   PRODUCT_TYPE[5].Motion.Gluing_Nozzle_Y.Position[20].Vel := 0;
   PRODUCT_TYPE[6].Motion.Gluing_Nozzle_Y.Position[20].Pos := 0.0;
   PRODUCT_TYPE[6].Motion.Gluing_Nozzle_Y.Position[20].Vel := 0;
   PRODUCT_TYPE[7].Motion.Gluing_Nozzle_Y.Position[20].Pos := 0.0;
   PRODUCT_TYPE[7].Motion.Gluing_Nozzle_Y.Position[20].Vel := 0;
   PRODUCT_TYPE[8].Motion.Gluing_Nozzle_Y.Position[20].Pos := 0.0;
   PRODUCT_TYPE[8].Motion.Gluing_Nozzle_Y.Position[20].Vel := 0;
   PRODUCT_TYPE[9].Motion.Gluing_Nozzle_Y.Position[20].Pos := 0.0;
   PRODUCT_TYPE[9].Motion.Gluing_Nozzle_Y.Position[20].Vel := 0;
   PRODUCT_TYPE[10].Motion.Gluing_Nozzle_Y.Position[20].Pos := 0.0;
   PRODUCT_TYPE[10].Motion.Gluing_Nozzle_Y.Position[20].Vel := 0;
   PRODUCT_TYPE[1].Motion.Ring_Turntable_Axis_1.Position[1].Pos := 3419;
   PRODUCT_TYPE[1].Motion.Ring_Turntable_Axis_1.Position[1].Vel := 10000;
   PRODUCT_TYPE[2].Motion.Ring_Turntable_Axis_1.Position[1].Pos := 3419;
   PRODUCT_TYPE[2].Motion.Ring_Turntable_Axis_1.Position[1].Vel := 10000;
   PRODUCT_TYPE[3].Motion.Ring_Turntable_Axis_1.Position[1].Pos := 3419;
   PRODUCT_TYPE[3].Motion.Ring_Turntable_Axis_1.Position[1].Vel := 10000;
   PRODUCT_TYPE[4].Motion.Ring_Turntable_Axis_1.Position[1].Pos := 3419;
   PRODUCT_TYPE[4].Motion.Ring_Turntable_Axis_1.Position[1].Vel := 10000;
   PRODUCT_TYPE[5].Motion.Ring_Turntable_Axis_1.Position[1].Pos := 3419;
   PRODUCT_TYPE[5].Motion.Ring_Turntable_Axis_1.Position[1].Vel := 10000;
   PRODUCT_TYPE[6].Motion.Ring_Turntable_Axis_1.Position[1].Pos := 3419;
   PRODUCT_TYPE[6].Motion.Ring_Turntable_Axis_1.Position[1].Vel := 10000;
   PRODUCT_TYPE[7].Motion.Ring_Turntable_Axis_1.Position[1].Pos := 3419;
   PRODUCT_TYPE[7].Motion.Ring_Turntable_Axis_1.Position[1].Vel := 10000;
   PRODUCT_TYPE[8].Motion.Ring_Turntable_Axis_1.Position[1].Pos := 3419;
   PRODUCT_TYPE[8].Motion.Ring_Turntable_Axis_1.Position[1].Vel := 10000;
   PRODUCT_TYPE[9].Motion.Ring_Turntable_Axis_1.Position[1].Pos := 3419;
   PRODUCT_TYPE[9].Motion.Ring_Turntable_Axis_1.Position[1].Vel := 10000;
   PRODUCT_TYPE[10].Motion.Ring_Turntable_Axis_1.Position[1].Pos := 3419;
   PRODUCT_TYPE[10].Motion.Ring_Turntable_Axis_1.Position[1].Vel := 10000;
   PRODUCT_TYPE[1].Motion.Ring_Turntable_Axis_1.Position[2].Pos := 48386;
   PRODUCT_TYPE[1].Motion.Ring_Turntable_Axis_1.Position[2].Vel := 10000;
   PRODUCT_TYPE[2].Motion.Ring_Turntable_Axis_1.Position[2].Pos := 48386;
   PRODUCT_TYPE[2].Motion.Ring_Turntable_Axis_1.Position[2].Vel := 10000;
   PRODUCT_TYPE[3].Motion.Ring_Turntable_Axis_1.Position[2].Pos := 48386;
   PRODUCT_TYPE[3].Motion.Ring_Turntable_Axis_1.Position[2].Vel := 10000;
   PRODUCT_TYPE[4].Motion.Ring_Turntable_Axis_1.Position[2].Pos := 48386;
   PRODUCT_TYPE[4].Motion.Ring_Turntable_Axis_1.Position[2].Vel := 10000;
   PRODUCT_TYPE[5].Motion.Ring_Turntable_Axis_1.Position[2].Pos := 48386;
   PRODUCT_TYPE[5].Motion.Ring_Turntable_Axis_1.Position[2].Vel := 10000;
   PRODUCT_TYPE[6].Motion.Ring_Turntable_Axis_1.Position[2].Pos := 48386;
   PRODUCT_TYPE[6].Motion.Ring_Turntable_Axis_1.Position[2].Vel := 10000;
   PRODUCT_TYPE[7].Motion.Ring_Turntable_Axis_1.Position[2].Pos := 48386;
   PRODUCT_TYPE[7].Motion.Ring_Turntable_Axis_1.Position[2].Vel := 10000;
   PRODUCT_TYPE[8].Motion.Ring_Turntable_Axis_1.Position[2].Pos := 48386;
   PRODUCT_TYPE[8].Motion.Ring_Turntable_Axis_1.Position[2].Vel := 10000;
   PRODUCT_TYPE[9].Motion.Ring_Turntable_Axis_1.Position[2].Pos := 48386;
   PRODUCT_TYPE[9].Motion.Ring_Turntable_Axis_1.Position[2].Vel := 10000;
   PRODUCT_TYPE[10].Motion.Ring_Turntable_Axis_1.Position[2].Pos := 48386;
   PRODUCT_TYPE[10].Motion.Ring_Turntable_Axis_1.Position[2].Vel := 10000;
   PRODUCT_TYPE[1].Motion.Ring_Turntable_Axis_1.Position[3].Pos := 93294;
   PRODUCT_TYPE[1].Motion.Ring_Turntable_Axis_1.Position[3].Vel := 10000;
   PRODUCT_TYPE[2].Motion.Ring_Turntable_Axis_1.Position[3].Pos := 93294;
   PRODUCT_TYPE[2].Motion.Ring_Turntable_Axis_1.Position[3].Vel := 10000;
   PRODUCT_TYPE[3].Motion.Ring_Turntable_Axis_1.Position[3].Pos := 93294;
   PRODUCT_TYPE[3].Motion.Ring_Turntable_Axis_1.Position[3].Vel := 10000;
   PRODUCT_TYPE[4].Motion.Ring_Turntable_Axis_1.Position[3].Pos := 93294;
   PRODUCT_TYPE[4].Motion.Ring_Turntable_Axis_1.Position[3].Vel := 10000;
   PRODUCT_TYPE[5].Motion.Ring_Turntable_Axis_1.Position[3].Pos := 93294;
   PRODUCT_TYPE[5].Motion.Ring_Turntable_Axis_1.Position[3].Vel := 10000;
   PRODUCT_TYPE[6].Motion.Ring_Turntable_Axis_1.Position[3].Pos := 93294;
   PRODUCT_TYPE[6].Motion.Ring_Turntable_Axis_1.Position[3].Vel := 10000;
   PRODUCT_TYPE[7].Motion.Ring_Turntable_Axis_1.Position[3].Pos := 93294;
   PRODUCT_TYPE[7].Motion.Ring_Turntable_Axis_1.Position[3].Vel := 10000;
   PRODUCT_TYPE[8].Motion.Ring_Turntable_Axis_1.Position[3].Pos := 93294;
   PRODUCT_TYPE[8].Motion.Ring_Turntable_Axis_1.Position[3].Vel := 10000;
   PRODUCT_TYPE[9].Motion.Ring_Turntable_Axis_1.Position[3].Pos := 93294;
   PRODUCT_TYPE[9].Motion.Ring_Turntable_Axis_1.Position[3].Vel := 10000;
   PRODUCT_TYPE[10].Motion.Ring_Turntable_Axis_1.Position[3].Pos := 93294;
   PRODUCT_TYPE[10].Motion.Ring_Turntable_Axis_1.Position[3].Vel := 10000;
   PRODUCT_TYPE[1].Motion.Ring_Turntable_Axis_1.Position[4].Pos := 138335;
   PRODUCT_TYPE[1].Motion.Ring_Turntable_Axis_1.Position[4].Vel := 10000;
   PRODUCT_TYPE[2].Motion.Ring_Turntable_Axis_1.Position[4].Pos := 138335;
   PRODUCT_TYPE[2].Motion.Ring_Turntable_Axis_1.Position[4].Vel := 10000;
   PRODUCT_TYPE[3].Motion.Ring_Turntable_Axis_1.Position[4].Pos := 138335;
   PRODUCT_TYPE[3].Motion.Ring_Turntable_Axis_1.Position[4].Vel := 10000;
   PRODUCT_TYPE[4].Motion.Ring_Turntable_Axis_1.Position[4].Pos := 138335;
   PRODUCT_TYPE[4].Motion.Ring_Turntable_Axis_1.Position[4].Vel := 10000;
   PRODUCT_TYPE[5].Motion.Ring_Turntable_Axis_1.Position[4].Pos := 138335;
   PRODUCT_TYPE[5].Motion.Ring_Turntable_Axis_1.Position[4].Vel := 10000;
   PRODUCT_TYPE[6].Motion.Ring_Turntable_Axis_1.Position[4].Pos := 138335;
   PRODUCT_TYPE[6].Motion.Ring_Turntable_Axis_1.Position[4].Vel := 10000;
   PRODUCT_TYPE[7].Motion.Ring_Turntable_Axis_1.Position[4].Pos := 138335;
   PRODUCT_TYPE[7].Motion.Ring_Turntable_Axis_1.Position[4].Vel := 10000;
   PRODUCT_TYPE[8].Motion.Ring_Turntable_Axis_1.Position[4].Pos := 138335;
   PRODUCT_TYPE[8].Motion.Ring_Turntable_Axis_1.Position[4].Vel := 10000;
   PRODUCT_TYPE[9].Motion.Ring_Turntable_Axis_1.Position[4].Pos := 138335;
   PRODUCT_TYPE[9].Motion.Ring_Turntable_Axis_1.Position[4].Vel := 10000;
   PRODUCT_TYPE[10].Motion.Ring_Turntable_Axis_1.Position[4].Pos := 138335;
   PRODUCT_TYPE[10].Motion.Ring_Turntable_Axis_1.Position[4].Vel := 10000;
   PRODUCT_TYPE[1].Motion.Ring_Turntable_Axis_1.Position[5].Pos := 183464;
   PRODUCT_TYPE[1].Motion.Ring_Turntable_Axis_1.Position[5].Vel := 10000;
   PRODUCT_TYPE[2].Motion.Ring_Turntable_Axis_1.Position[5].Pos := 183464;
   PRODUCT_TYPE[2].Motion.Ring_Turntable_Axis_1.Position[5].Vel := 10000;
   PRODUCT_TYPE[3].Motion.Ring_Turntable_Axis_1.Position[5].Pos := 183464;
   PRODUCT_TYPE[3].Motion.Ring_Turntable_Axis_1.Position[5].Vel := 10000;
   PRODUCT_TYPE[4].Motion.Ring_Turntable_Axis_1.Position[5].Pos := 183464;
   PRODUCT_TYPE[4].Motion.Ring_Turntable_Axis_1.Position[5].Vel := 10000;
   PRODUCT_TYPE[5].Motion.Ring_Turntable_Axis_1.Position[5].Pos := 183464;
   PRODUCT_TYPE[5].Motion.Ring_Turntable_Axis_1.Position[5].Vel := 10000;
   PRODUCT_TYPE[6].Motion.Ring_Turntable_Axis_1.Position[5].Pos := 183464;
   PRODUCT_TYPE[6].Motion.Ring_Turntable_Axis_1.Position[5].Vel := 10000;
   PRODUCT_TYPE[7].Motion.Ring_Turntable_Axis_1.Position[5].Pos := 183464;
   PRODUCT_TYPE[7].Motion.Ring_Turntable_Axis_1.Position[5].Vel := 10000;
   PRODUCT_TYPE[8].Motion.Ring_Turntable_Axis_1.Position[5].Pos := 183464;
   PRODUCT_TYPE[8].Motion.Ring_Turntable_Axis_1.Position[5].Vel := 10000;
   PRODUCT_TYPE[9].Motion.Ring_Turntable_Axis_1.Position[5].Pos := 183464;
   PRODUCT_TYPE[9].Motion.Ring_Turntable_Axis_1.Position[5].Vel := 10000;
   PRODUCT_TYPE[10].Motion.Ring_Turntable_Axis_1.Position[5].Pos := 183464;
   PRODUCT_TYPE[10].Motion.Ring_Turntable_Axis_1.Position[5].Vel := 10000;
   PRODUCT_TYPE[1].Motion.Ring_Turntable_Axis_1.Position[6].Pos := 228443;
   PRODUCT_TYPE[1].Motion.Ring_Turntable_Axis_1.Position[6].Vel := 10000;
   PRODUCT_TYPE[2].Motion.Ring_Turntable_Axis_1.Position[6].Pos := 228443;
   PRODUCT_TYPE[2].Motion.Ring_Turntable_Axis_1.Position[6].Vel := 10000;
   PRODUCT_TYPE[3].Motion.Ring_Turntable_Axis_1.Position[6].Pos := 228443;
   PRODUCT_TYPE[3].Motion.Ring_Turntable_Axis_1.Position[6].Vel := 10000;
   PRODUCT_TYPE[4].Motion.Ring_Turntable_Axis_1.Position[6].Pos := 228443;
   PRODUCT_TYPE[4].Motion.Ring_Turntable_Axis_1.Position[6].Vel := 10000;
   PRODUCT_TYPE[5].Motion.Ring_Turntable_Axis_1.Position[6].Pos := 228443;
   PRODUCT_TYPE[5].Motion.Ring_Turntable_Axis_1.Position[6].Vel := 10000;
   PRODUCT_TYPE[6].Motion.Ring_Turntable_Axis_1.Position[6].Pos := 228443;
   PRODUCT_TYPE[6].Motion.Ring_Turntable_Axis_1.Position[6].Vel := 10000;
   PRODUCT_TYPE[7].Motion.Ring_Turntable_Axis_1.Position[6].Pos := 228443;
   PRODUCT_TYPE[7].Motion.Ring_Turntable_Axis_1.Position[6].Vel := 10000;
   PRODUCT_TYPE[8].Motion.Ring_Turntable_Axis_1.Position[6].Pos := 228443;
   PRODUCT_TYPE[8].Motion.Ring_Turntable_Axis_1.Position[6].Vel := 10000;
   PRODUCT_TYPE[9].Motion.Ring_Turntable_Axis_1.Position[6].Pos := 228443;
   PRODUCT_TYPE[9].Motion.Ring_Turntable_Axis_1.Position[6].Vel := 10000;
   PRODUCT_TYPE[10].Motion.Ring_Turntable_Axis_1.Position[6].Pos := 228443;
   PRODUCT_TYPE[10].Motion.Ring_Turntable_Axis_1.Position[6].Vel := 10000;
   PRODUCT_TYPE[1].Motion.Ring_Turntable_Axis_1.Position[7].Pos := 273535;
   PRODUCT_TYPE[1].Motion.Ring_Turntable_Axis_1.Position[7].Vel := 10000;
   PRODUCT_TYPE[2].Motion.Ring_Turntable_Axis_1.Position[7].Pos := 273535;
   PRODUCT_TYPE[2].Motion.Ring_Turntable_Axis_1.Position[7].Vel := 10000;
   PRODUCT_TYPE[3].Motion.Ring_Turntable_Axis_1.Position[7].Pos := 273535;
   PRODUCT_TYPE[3].Motion.Ring_Turntable_Axis_1.Position[7].Vel := 10000;
   PRODUCT_TYPE[4].Motion.Ring_Turntable_Axis_1.Position[7].Pos := 273535;
   PRODUCT_TYPE[4].Motion.Ring_Turntable_Axis_1.Position[7].Vel := 10000;
   PRODUCT_TYPE[5].Motion.Ring_Turntable_Axis_1.Position[7].Pos := 273535;
   PRODUCT_TYPE[5].Motion.Ring_Turntable_Axis_1.Position[7].Vel := 10000;
   PRODUCT_TYPE[6].Motion.Ring_Turntable_Axis_1.Position[7].Pos := 273535;
   PRODUCT_TYPE[6].Motion.Ring_Turntable_Axis_1.Position[7].Vel := 10000;
   PRODUCT_TYPE[7].Motion.Ring_Turntable_Axis_1.Position[7].Pos := 273535;
   PRODUCT_TYPE[7].Motion.Ring_Turntable_Axis_1.Position[7].Vel := 10000;
   PRODUCT_TYPE[8].Motion.Ring_Turntable_Axis_1.Position[7].Pos := 273535;
   PRODUCT_TYPE[8].Motion.Ring_Turntable_Axis_1.Position[7].Vel := 10000;
   PRODUCT_TYPE[9].Motion.Ring_Turntable_Axis_1.Position[7].Pos := 273535;
   PRODUCT_TYPE[9].Motion.Ring_Turntable_Axis_1.Position[7].Vel := 10000;
   PRODUCT_TYPE[10].Motion.Ring_Turntable_Axis_1.Position[7].Pos := 273535;
   PRODUCT_TYPE[10].Motion.Ring_Turntable_Axis_1.Position[7].Vel := 10000;
   PRODUCT_TYPE[1].Motion.Ring_Turntable_Axis_1.Position[8].Pos := 318250;
   PRODUCT_TYPE[1].Motion.Ring_Turntable_Axis_1.Position[8].Vel := 10000;
   PRODUCT_TYPE[2].Motion.Ring_Turntable_Axis_1.Position[8].Pos := 318250;
   PRODUCT_TYPE[2].Motion.Ring_Turntable_Axis_1.Position[8].Vel := 10000;
   PRODUCT_TYPE[3].Motion.Ring_Turntable_Axis_1.Position[8].Pos := 318250;
   PRODUCT_TYPE[3].Motion.Ring_Turntable_Axis_1.Position[8].Vel := 10000;
   PRODUCT_TYPE[4].Motion.Ring_Turntable_Axis_1.Position[8].Pos := 318250;
   PRODUCT_TYPE[4].Motion.Ring_Turntable_Axis_1.Position[8].Vel := 10000;
   PRODUCT_TYPE[5].Motion.Ring_Turntable_Axis_1.Position[8].Pos := 318250;
   PRODUCT_TYPE[5].Motion.Ring_Turntable_Axis_1.Position[8].Vel := 10000;
   PRODUCT_TYPE[6].Motion.Ring_Turntable_Axis_1.Position[8].Pos := 318250;
   PRODUCT_TYPE[6].Motion.Ring_Turntable_Axis_1.Position[8].Vel := 10000;
   PRODUCT_TYPE[7].Motion.Ring_Turntable_Axis_1.Position[8].Pos := 318250;
   PRODUCT_TYPE[7].Motion.Ring_Turntable_Axis_1.Position[8].Vel := 10000;
   PRODUCT_TYPE[8].Motion.Ring_Turntable_Axis_1.Position[8].Pos := 318250;
   PRODUCT_TYPE[8].Motion.Ring_Turntable_Axis_1.Position[8].Vel := 10000;
   PRODUCT_TYPE[9].Motion.Ring_Turntable_Axis_1.Position[8].Pos := 318250;
   PRODUCT_TYPE[9].Motion.Ring_Turntable_Axis_1.Position[8].Vel := 10000;
   PRODUCT_TYPE[10].Motion.Ring_Turntable_Axis_1.Position[8].Pos := 318250;
   PRODUCT_TYPE[10].Motion.Ring_Turntable_Axis_1.Position[8].Vel := 10000;
   PRODUCT_TYPE[1].Motion.Ring_Turntable_Axis_1.Position[9].Pos := 0;
   PRODUCT_TYPE[1].Motion.Ring_Turntable_Axis_1.Position[9].Vel := 0;
   PRODUCT_TYPE[2].Motion.Ring_Turntable_Axis_1.Position[9].Pos := 0;
   PRODUCT_TYPE[2].Motion.Ring_Turntable_Axis_1.Position[9].Vel := 0;
   PRODUCT_TYPE[3].Motion.Ring_Turntable_Axis_1.Position[9].Pos := 0;
   PRODUCT_TYPE[3].Motion.Ring_Turntable_Axis_1.Position[9].Vel := 0;
   PRODUCT_TYPE[4].Motion.Ring_Turntable_Axis_1.Position[9].Pos := 0;
   PRODUCT_TYPE[4].Motion.Ring_Turntable_Axis_1.Position[9].Vel := 0;
   PRODUCT_TYPE[5].Motion.Ring_Turntable_Axis_1.Position[9].Pos := 0;
   PRODUCT_TYPE[5].Motion.Ring_Turntable_Axis_1.Position[9].Vel := 0;
   PRODUCT_TYPE[6].Motion.Ring_Turntable_Axis_1.Position[9].Pos := 0;
   PRODUCT_TYPE[6].Motion.Ring_Turntable_Axis_1.Position[9].Vel := 0;
   PRODUCT_TYPE[7].Motion.Ring_Turntable_Axis_1.Position[9].Pos := 0;
   PRODUCT_TYPE[7].Motion.Ring_Turntable_Axis_1.Position[9].Vel := 0;
   PRODUCT_TYPE[8].Motion.Ring_Turntable_Axis_1.Position[9].Pos := 0;
   PRODUCT_TYPE[8].Motion.Ring_Turntable_Axis_1.Position[9].Vel := 0;
   PRODUCT_TYPE[9].Motion.Ring_Turntable_Axis_1.Position[9].Pos := 0;
   PRODUCT_TYPE[9].Motion.Ring_Turntable_Axis_1.Position[9].Vel := 0;
   PRODUCT_TYPE[10].Motion.Ring_Turntable_Axis_1.Position[9].Pos := 0;
   PRODUCT_TYPE[10].Motion.Ring_Turntable_Axis_1.Position[9].Vel := 0;
   PRODUCT_TYPE[1].Motion.Ring_Turntable_Axis_1.Position[10].Pos := 0;
   PRODUCT_TYPE[1].Motion.Ring_Turntable_Axis_1.Position[10].Vel := 0;
   PRODUCT_TYPE[2].Motion.Ring_Turntable_Axis_1.Position[10].Pos := 0;
   PRODUCT_TYPE[2].Motion.Ring_Turntable_Axis_1.Position[10].Vel := 0;
   PRODUCT_TYPE[3].Motion.Ring_Turntable_Axis_1.Position[10].Pos := 0;
   PRODUCT_TYPE[3].Motion.Ring_Turntable_Axis_1.Position[10].Vel := 0;
   PRODUCT_TYPE[4].Motion.Ring_Turntable_Axis_1.Position[10].Pos := 0;
   PRODUCT_TYPE[4].Motion.Ring_Turntable_Axis_1.Position[10].Vel := 0;
   PRODUCT_TYPE[5].Motion.Ring_Turntable_Axis_1.Position[10].Pos := 0;
   PRODUCT_TYPE[5].Motion.Ring_Turntable_Axis_1.Position[10].Vel := 0;
   PRODUCT_TYPE[6].Motion.Ring_Turntable_Axis_1.Position[10].Pos := 0;
   PRODUCT_TYPE[6].Motion.Ring_Turntable_Axis_1.Position[10].Vel := 0;
   PRODUCT_TYPE[7].Motion.Ring_Turntable_Axis_1.Position[10].Pos := 0;
   PRODUCT_TYPE[7].Motion.Ring_Turntable_Axis_1.Position[10].Vel := 0;
   PRODUCT_TYPE[8].Motion.Ring_Turntable_Axis_1.Position[10].Pos := 0;
   PRODUCT_TYPE[8].Motion.Ring_Turntable_Axis_1.Position[10].Vel := 0;
   PRODUCT_TYPE[9].Motion.Ring_Turntable_Axis_1.Position[10].Pos := 0;
   PRODUCT_TYPE[9].Motion.Ring_Turntable_Axis_1.Position[10].Vel := 0;
   PRODUCT_TYPE[10].Motion.Ring_Turntable_Axis_1.Position[10].Pos := 0;
   PRODUCT_TYPE[10].Motion.Ring_Turntable_Axis_1.Position[10].Vel := 0;
   PRODUCT_TYPE[1].Motion.Ring_Turntable_Axis_1.Position[11].Pos := 0;
   PRODUCT_TYPE[1].Motion.Ring_Turntable_Axis_1.Position[11].Vel := 0;
   PRODUCT_TYPE[2].Motion.Ring_Turntable_Axis_1.Position[11].Pos := 0;
   PRODUCT_TYPE[2].Motion.Ring_Turntable_Axis_1.Position[11].Vel := 0;
   PRODUCT_TYPE[3].Motion.Ring_Turntable_Axis_1.Position[11].Pos := 0;
   PRODUCT_TYPE[3].Motion.Ring_Turntable_Axis_1.Position[11].Vel := 0;
   PRODUCT_TYPE[4].Motion.Ring_Turntable_Axis_1.Position[11].Pos := 0;
   PRODUCT_TYPE[4].Motion.Ring_Turntable_Axis_1.Position[11].Vel := 0;
   PRODUCT_TYPE[5].Motion.Ring_Turntable_Axis_1.Position[11].Pos := 0;
   PRODUCT_TYPE[5].Motion.Ring_Turntable_Axis_1.Position[11].Vel := 0;
   PRODUCT_TYPE[6].Motion.Ring_Turntable_Axis_1.Position[11].Pos := 0;
   PRODUCT_TYPE[6].Motion.Ring_Turntable_Axis_1.Position[11].Vel := 0;
   PRODUCT_TYPE[7].Motion.Ring_Turntable_Axis_1.Position[11].Pos := 0;
   PRODUCT_TYPE[7].Motion.Ring_Turntable_Axis_1.Position[11].Vel := 0;
   PRODUCT_TYPE[8].Motion.Ring_Turntable_Axis_1.Position[11].Pos := 0;
   PRODUCT_TYPE[8].Motion.Ring_Turntable_Axis_1.Position[11].Vel := 0;
   PRODUCT_TYPE[9].Motion.Ring_Turntable_Axis_1.Position[11].Pos := 0;
   PRODUCT_TYPE[9].Motion.Ring_Turntable_Axis_1.Position[11].Vel := 0;
   PRODUCT_TYPE[10].Motion.Ring_Turntable_Axis_1.Position[11].Pos := 0;
   PRODUCT_TYPE[10].Motion.Ring_Turntable_Axis_1.Position[11].Vel := 0;
   PRODUCT_TYPE[1].Motion.Ring_Turntable_Axis_1.Position[12].Pos := 0;
   PRODUCT_TYPE[1].Motion.Ring_Turntable_Axis_1.Position[12].Vel := 0;
   PRODUCT_TYPE[2].Motion.Ring_Turntable_Axis_1.Position[12].Pos := 0;
   PRODUCT_TYPE[2].Motion.Ring_Turntable_Axis_1.Position[12].Vel := 0;
   PRODUCT_TYPE[3].Motion.Ring_Turntable_Axis_1.Position[12].Pos := 0;
   PRODUCT_TYPE[3].Motion.Ring_Turntable_Axis_1.Position[12].Vel := 0;
   PRODUCT_TYPE[4].Motion.Ring_Turntable_Axis_1.Position[12].Pos := 0;
   PRODUCT_TYPE[4].Motion.Ring_Turntable_Axis_1.Position[12].Vel := 0;
   PRODUCT_TYPE[5].Motion.Ring_Turntable_Axis_1.Position[12].Pos := 0;
   PRODUCT_TYPE[5].Motion.Ring_Turntable_Axis_1.Position[12].Vel := 0;
   PRODUCT_TYPE[6].Motion.Ring_Turntable_Axis_1.Position[12].Pos := 0;
   PRODUCT_TYPE[6].Motion.Ring_Turntable_Axis_1.Position[12].Vel := 0;
   PRODUCT_TYPE[7].Motion.Ring_Turntable_Axis_1.Position[12].Pos := 0;
   PRODUCT_TYPE[7].Motion.Ring_Turntable_Axis_1.Position[12].Vel := 0;
   PRODUCT_TYPE[8].Motion.Ring_Turntable_Axis_1.Position[12].Pos := 0;
   PRODUCT_TYPE[8].Motion.Ring_Turntable_Axis_1.Position[12].Vel := 0;
   PRODUCT_TYPE[9].Motion.Ring_Turntable_Axis_1.Position[12].Pos := 0;
   PRODUCT_TYPE[9].Motion.Ring_Turntable_Axis_1.Position[12].Vel := 0;
   PRODUCT_TYPE[10].Motion.Ring_Turntable_Axis_1.Position[12].Pos := 0;
   PRODUCT_TYPE[10].Motion.Ring_Turntable_Axis_1.Position[12].Vel := 0;
   PRODUCT_TYPE[1].Motion.Ring_Turntable_Axis_1.Position[13].Pos := 0;
   PRODUCT_TYPE[1].Motion.Ring_Turntable_Axis_1.Position[13].Vel := 0;
   PRODUCT_TYPE[2].Motion.Ring_Turntable_Axis_1.Position[13].Pos := 0;
   PRODUCT_TYPE[2].Motion.Ring_Turntable_Axis_1.Position[13].Vel := 0;
   PRODUCT_TYPE[3].Motion.Ring_Turntable_Axis_1.Position[13].Pos := 0;
   PRODUCT_TYPE[3].Motion.Ring_Turntable_Axis_1.Position[13].Vel := 0;
   PRODUCT_TYPE[4].Motion.Ring_Turntable_Axis_1.Position[13].Pos := 0;
   PRODUCT_TYPE[4].Motion.Ring_Turntable_Axis_1.Position[13].Vel := 0;
   PRODUCT_TYPE[5].Motion.Ring_Turntable_Axis_1.Position[13].Pos := 0;
   PRODUCT_TYPE[5].Motion.Ring_Turntable_Axis_1.Position[13].Vel := 0;
   PRODUCT_TYPE[6].Motion.Ring_Turntable_Axis_1.Position[13].Pos := 0;
   PRODUCT_TYPE[6].Motion.Ring_Turntable_Axis_1.Position[13].Vel := 0;
   PRODUCT_TYPE[7].Motion.Ring_Turntable_Axis_1.Position[13].Pos := 0;
   PRODUCT_TYPE[7].Motion.Ring_Turntable_Axis_1.Position[13].Vel := 0;
   PRODUCT_TYPE[8].Motion.Ring_Turntable_Axis_1.Position[13].Pos := 0;
   PRODUCT_TYPE[8].Motion.Ring_Turntable_Axis_1.Position[13].Vel := 0;
   PRODUCT_TYPE[9].Motion.Ring_Turntable_Axis_1.Position[13].Pos := 0;
   PRODUCT_TYPE[9].Motion.Ring_Turntable_Axis_1.Position[13].Vel := 0;
   PRODUCT_TYPE[10].Motion.Ring_Turntable_Axis_1.Position[13].Pos := 0;
   PRODUCT_TYPE[10].Motion.Ring_Turntable_Axis_1.Position[13].Vel := 0;
   PRODUCT_TYPE[1].Motion.Ring_Turntable_Axis_1.Position[14].Pos := 0;
   PRODUCT_TYPE[1].Motion.Ring_Turntable_Axis_1.Position[14].Vel := 0;
   PRODUCT_TYPE[2].Motion.Ring_Turntable_Axis_1.Position[14].Pos := 0;
   PRODUCT_TYPE[2].Motion.Ring_Turntable_Axis_1.Position[14].Vel := 0;
   PRODUCT_TYPE[3].Motion.Ring_Turntable_Axis_1.Position[14].Pos := 0;
   PRODUCT_TYPE[3].Motion.Ring_Turntable_Axis_1.Position[14].Vel := 0;
   PRODUCT_TYPE[4].Motion.Ring_Turntable_Axis_1.Position[14].Pos := 0;
   PRODUCT_TYPE[4].Motion.Ring_Turntable_Axis_1.Position[14].Vel := 0;
   PRODUCT_TYPE[5].Motion.Ring_Turntable_Axis_1.Position[14].Pos := 0;
   PRODUCT_TYPE[5].Motion.Ring_Turntable_Axis_1.Position[14].Vel := 0;
   PRODUCT_TYPE[6].Motion.Ring_Turntable_Axis_1.Position[14].Pos := 0;
   PRODUCT_TYPE[6].Motion.Ring_Turntable_Axis_1.Position[14].Vel := 0;
   PRODUCT_TYPE[7].Motion.Ring_Turntable_Axis_1.Position[14].Pos := 0;
   PRODUCT_TYPE[7].Motion.Ring_Turntable_Axis_1.Position[14].Vel := 0;
   PRODUCT_TYPE[8].Motion.Ring_Turntable_Axis_1.Position[14].Pos := 0;
   PRODUCT_TYPE[8].Motion.Ring_Turntable_Axis_1.Position[14].Vel := 0;
   PRODUCT_TYPE[9].Motion.Ring_Turntable_Axis_1.Position[14].Pos := 0;
   PRODUCT_TYPE[9].Motion.Ring_Turntable_Axis_1.Position[14].Vel := 0;
   PRODUCT_TYPE[10].Motion.Ring_Turntable_Axis_1.Position[14].Pos := 0;
   PRODUCT_TYPE[10].Motion.Ring_Turntable_Axis_1.Position[14].Vel := 0;
   PRODUCT_TYPE[1].Motion.Ring_Turntable_Axis_1.Position[15].Pos := 0;
   PRODUCT_TYPE[1].Motion.Ring_Turntable_Axis_1.Position[15].Vel := 0;
   PRODUCT_TYPE[2].Motion.Ring_Turntable_Axis_1.Position[15].Pos := 0;
   PRODUCT_TYPE[2].Motion.Ring_Turntable_Axis_1.Position[15].Vel := 0;
   PRODUCT_TYPE[3].Motion.Ring_Turntable_Axis_1.Position[15].Pos := 0;
   PRODUCT_TYPE[3].Motion.Ring_Turntable_Axis_1.Position[15].Vel := 0;
   PRODUCT_TYPE[4].Motion.Ring_Turntable_Axis_1.Position[15].Pos := 0;
   PRODUCT_TYPE[4].Motion.Ring_Turntable_Axis_1.Position[15].Vel := 0;
   PRODUCT_TYPE[5].Motion.Ring_Turntable_Axis_1.Position[15].Pos := 0;
   PRODUCT_TYPE[5].Motion.Ring_Turntable_Axis_1.Position[15].Vel := 0;
   PRODUCT_TYPE[6].Motion.Ring_Turntable_Axis_1.Position[15].Pos := 0;
   PRODUCT_TYPE[6].Motion.Ring_Turntable_Axis_1.Position[15].Vel := 0;
   PRODUCT_TYPE[7].Motion.Ring_Turntable_Axis_1.Position[15].Pos := 0;
   PRODUCT_TYPE[7].Motion.Ring_Turntable_Axis_1.Position[15].Vel := 0;
   PRODUCT_TYPE[8].Motion.Ring_Turntable_Axis_1.Position[15].Pos := 0;
   PRODUCT_TYPE[8].Motion.Ring_Turntable_Axis_1.Position[15].Vel := 0;
   PRODUCT_TYPE[9].Motion.Ring_Turntable_Axis_1.Position[15].Pos := 0;
   PRODUCT_TYPE[9].Motion.Ring_Turntable_Axis_1.Position[15].Vel := 0;
   PRODUCT_TYPE[10].Motion.Ring_Turntable_Axis_1.Position[15].Pos := 0;
   PRODUCT_TYPE[10].Motion.Ring_Turntable_Axis_1.Position[15].Vel := 0;
   PRODUCT_TYPE[1].Motion.Ring_Turntable_Axis_1.Position[16].Pos := 0;
   PRODUCT_TYPE[1].Motion.Ring_Turntable_Axis_1.Position[16].Vel := 0;
   PRODUCT_TYPE[2].Motion.Ring_Turntable_Axis_1.Position[16].Pos := 0;
   PRODUCT_TYPE[2].Motion.Ring_Turntable_Axis_1.Position[16].Vel := 0;
   PRODUCT_TYPE[3].Motion.Ring_Turntable_Axis_1.Position[16].Pos := 0;
   PRODUCT_TYPE[3].Motion.Ring_Turntable_Axis_1.Position[16].Vel := 0;
   PRODUCT_TYPE[4].Motion.Ring_Turntable_Axis_1.Position[16].Pos := 0;
   PRODUCT_TYPE[4].Motion.Ring_Turntable_Axis_1.Position[16].Vel := 0;
   PRODUCT_TYPE[5].Motion.Ring_Turntable_Axis_1.Position[16].Pos := 0;
   PRODUCT_TYPE[5].Motion.Ring_Turntable_Axis_1.Position[16].Vel := 0;
   PRODUCT_TYPE[6].Motion.Ring_Turntable_Axis_1.Position[16].Pos := 0;
   PRODUCT_TYPE[6].Motion.Ring_Turntable_Axis_1.Position[16].Vel := 0;
   PRODUCT_TYPE[7].Motion.Ring_Turntable_Axis_1.Position[16].Pos := 0;
   PRODUCT_TYPE[7].Motion.Ring_Turntable_Axis_1.Position[16].Vel := 0;
   PRODUCT_TYPE[8].Motion.Ring_Turntable_Axis_1.Position[16].Pos := 0;
   PRODUCT_TYPE[8].Motion.Ring_Turntable_Axis_1.Position[16].Vel := 0;
   PRODUCT_TYPE[9].Motion.Ring_Turntable_Axis_1.Position[16].Pos := 0;
   PRODUCT_TYPE[9].Motion.Ring_Turntable_Axis_1.Position[16].Vel := 0;
   PRODUCT_TYPE[10].Motion.Ring_Turntable_Axis_1.Position[16].Pos := 0;
   PRODUCT_TYPE[10].Motion.Ring_Turntable_Axis_1.Position[16].Vel := 0;
   PRODUCT_TYPE[1].Motion.Ring_Turntable_Axis_1.Position[17].Pos := 0;
   PRODUCT_TYPE[1].Motion.Ring_Turntable_Axis_1.Position[17].Vel := 0;
   PRODUCT_TYPE[2].Motion.Ring_Turntable_Axis_1.Position[17].Pos := 0;
   PRODUCT_TYPE[2].Motion.Ring_Turntable_Axis_1.Position[17].Vel := 0;
   PRODUCT_TYPE[3].Motion.Ring_Turntable_Axis_1.Position[17].Pos := 0;
   PRODUCT_TYPE[3].Motion.Ring_Turntable_Axis_1.Position[17].Vel := 0;
   PRODUCT_TYPE[4].Motion.Ring_Turntable_Axis_1.Position[17].Pos := 0;
   PRODUCT_TYPE[4].Motion.Ring_Turntable_Axis_1.Position[17].Vel := 0;
   PRODUCT_TYPE[5].Motion.Ring_Turntable_Axis_1.Position[17].Pos := 0;
   PRODUCT_TYPE[5].Motion.Ring_Turntable_Axis_1.Position[17].Vel := 0;
   PRODUCT_TYPE[6].Motion.Ring_Turntable_Axis_1.Position[17].Pos := 0;
   PRODUCT_TYPE[6].Motion.Ring_Turntable_Axis_1.Position[17].Vel := 0;
   PRODUCT_TYPE[7].Motion.Ring_Turntable_Axis_1.Position[17].Pos := 0;
   PRODUCT_TYPE[7].Motion.Ring_Turntable_Axis_1.Position[17].Vel := 0;
   PRODUCT_TYPE[8].Motion.Ring_Turntable_Axis_1.Position[17].Pos := 0;
   PRODUCT_TYPE[8].Motion.Ring_Turntable_Axis_1.Position[17].Vel := 0;
   PRODUCT_TYPE[9].Motion.Ring_Turntable_Axis_1.Position[17].Pos := 0;
   PRODUCT_TYPE[9].Motion.Ring_Turntable_Axis_1.Position[17].Vel := 0;
   PRODUCT_TYPE[10].Motion.Ring_Turntable_Axis_1.Position[17].Pos := 0;
   PRODUCT_TYPE[10].Motion.Ring_Turntable_Axis_1.Position[17].Vel := 0;
   PRODUCT_TYPE[1].Motion.Ring_Turntable_Axis_1.Position[18].Pos := 0;
   PRODUCT_TYPE[1].Motion.Ring_Turntable_Axis_1.Position[18].Vel := 0;
   PRODUCT_TYPE[2].Motion.Ring_Turntable_Axis_1.Position[18].Pos := 0;
   PRODUCT_TYPE[2].Motion.Ring_Turntable_Axis_1.Position[18].Vel := 0;
   PRODUCT_TYPE[3].Motion.Ring_Turntable_Axis_1.Position[18].Pos := 0;
   PRODUCT_TYPE[3].Motion.Ring_Turntable_Axis_1.Position[18].Vel := 0;
   PRODUCT_TYPE[4].Motion.Ring_Turntable_Axis_1.Position[18].Pos := 0;
   PRODUCT_TYPE[4].Motion.Ring_Turntable_Axis_1.Position[18].Vel := 0;
   PRODUCT_TYPE[5].Motion.Ring_Turntable_Axis_1.Position[18].Pos := 0;
   PRODUCT_TYPE[5].Motion.Ring_Turntable_Axis_1.Position[18].Vel := 0;
   PRODUCT_TYPE[6].Motion.Ring_Turntable_Axis_1.Position[18].Pos := 0;
   PRODUCT_TYPE[6].Motion.Ring_Turntable_Axis_1.Position[18].Vel := 0;
   PRODUCT_TYPE[7].Motion.Ring_Turntable_Axis_1.Position[18].Pos := 0;
   PRODUCT_TYPE[7].Motion.Ring_Turntable_Axis_1.Position[18].Vel := 0;
   PRODUCT_TYPE[8].Motion.Ring_Turntable_Axis_1.Position[18].Pos := 0;
   PRODUCT_TYPE[8].Motion.Ring_Turntable_Axis_1.Position[18].Vel := 0;
   PRODUCT_TYPE[9].Motion.Ring_Turntable_Axis_1.Position[18].Pos := 0;
   PRODUCT_TYPE[9].Motion.Ring_Turntable_Axis_1.Position[18].Vel := 0;
   PRODUCT_TYPE[10].Motion.Ring_Turntable_Axis_1.Position[18].Pos := 0;
   PRODUCT_TYPE[10].Motion.Ring_Turntable_Axis_1.Position[18].Vel := 0;
   PRODUCT_TYPE[1].Motion.Ring_Turntable_Axis_1.Position[19].Pos := 0;
   PRODUCT_TYPE[1].Motion.Ring_Turntable_Axis_1.Position[19].Vel := 0;
   PRODUCT_TYPE[2].Motion.Ring_Turntable_Axis_1.Position[19].Pos := 0;
   PRODUCT_TYPE[2].Motion.Ring_Turntable_Axis_1.Position[19].Vel := 0;
   PRODUCT_TYPE[3].Motion.Ring_Turntable_Axis_1.Position[19].Pos := 0;
   PRODUCT_TYPE[3].Motion.Ring_Turntable_Axis_1.Position[19].Vel := 0;
   PRODUCT_TYPE[4].Motion.Ring_Turntable_Axis_1.Position[19].Pos := 0;
   PRODUCT_TYPE[4].Motion.Ring_Turntable_Axis_1.Position[19].Vel := 0;
   PRODUCT_TYPE[5].Motion.Ring_Turntable_Axis_1.Position[19].Pos := 0;
   PRODUCT_TYPE[5].Motion.Ring_Turntable_Axis_1.Position[19].Vel := 0;
   PRODUCT_TYPE[6].Motion.Ring_Turntable_Axis_1.Position[19].Pos := 0;
   PRODUCT_TYPE[6].Motion.Ring_Turntable_Axis_1.Position[19].Vel := 0;
   PRODUCT_TYPE[7].Motion.Ring_Turntable_Axis_1.Position[19].Pos := 0;
   PRODUCT_TYPE[7].Motion.Ring_Turntable_Axis_1.Position[19].Vel := 0;
   PRODUCT_TYPE[8].Motion.Ring_Turntable_Axis_1.Position[19].Pos := 0;
   PRODUCT_TYPE[8].Motion.Ring_Turntable_Axis_1.Position[19].Vel := 0;
   PRODUCT_TYPE[9].Motion.Ring_Turntable_Axis_1.Position[19].Pos := 0;
   PRODUCT_TYPE[9].Motion.Ring_Turntable_Axis_1.Position[19].Vel := 0;
   PRODUCT_TYPE[10].Motion.Ring_Turntable_Axis_1.Position[19].Pos := 0;
   PRODUCT_TYPE[10].Motion.Ring_Turntable_Axis_1.Position[19].Vel := 0;
   PRODUCT_TYPE[1].Motion.Ring_Turntable_Axis_1.Position[20].Pos := 0;
   PRODUCT_TYPE[1].Motion.Ring_Turntable_Axis_1.Position[20].Vel := 0;
   PRODUCT_TYPE[2].Motion.Ring_Turntable_Axis_1.Position[20].Pos := 0;
   PRODUCT_TYPE[2].Motion.Ring_Turntable_Axis_1.Position[20].Vel := 0;
   PRODUCT_TYPE[3].Motion.Ring_Turntable_Axis_1.Position[20].Pos := 0;
   PRODUCT_TYPE[3].Motion.Ring_Turntable_Axis_1.Position[20].Vel := 0;
   PRODUCT_TYPE[4].Motion.Ring_Turntable_Axis_1.Position[20].Pos := 0;
   PRODUCT_TYPE[4].Motion.Ring_Turntable_Axis_1.Position[20].Vel := 0;
   PRODUCT_TYPE[5].Motion.Ring_Turntable_Axis_1.Position[20].Pos := 0;
   PRODUCT_TYPE[5].Motion.Ring_Turntable_Axis_1.Position[20].Vel := 0;
   PRODUCT_TYPE[6].Motion.Ring_Turntable_Axis_1.Position[20].Pos := 0;
   PRODUCT_TYPE[6].Motion.Ring_Turntable_Axis_1.Position[20].Vel := 0;
   PRODUCT_TYPE[7].Motion.Ring_Turntable_Axis_1.Position[20].Pos := 0;
   PRODUCT_TYPE[7].Motion.Ring_Turntable_Axis_1.Position[20].Vel := 0;
   PRODUCT_TYPE[8].Motion.Ring_Turntable_Axis_1.Position[20].Pos := 0;
   PRODUCT_TYPE[8].Motion.Ring_Turntable_Axis_1.Position[20].Vel := 0;
   PRODUCT_TYPE[9].Motion.Ring_Turntable_Axis_1.Position[20].Pos := 0;
   PRODUCT_TYPE[9].Motion.Ring_Turntable_Axis_1.Position[20].Vel := 0;
   PRODUCT_TYPE[10].Motion.Ring_Turntable_Axis_1.Position[20].Pos := 0;
   PRODUCT_TYPE[10].Motion.Ring_Turntable_Axis_1.Position[20].Vel := 0;
   PRODUCT_TYPE[1].Motion.Shaft_Scan_Turntable_Axis.Position[1].Pos := 0;
   PRODUCT_TYPE[1].Motion.Shaft_Scan_Turntable_Axis.Position[1].Vel := 10000;
   PRODUCT_TYPE[2].Motion.Shaft_Scan_Turntable_Axis.Position[1].Pos := 0;
   PRODUCT_TYPE[2].Motion.Shaft_Scan_Turntable_Axis.Position[1].Vel := 10000;
   PRODUCT_TYPE[3].Motion.Shaft_Scan_Turntable_Axis.Position[1].Pos := 0;
   PRODUCT_TYPE[3].Motion.Shaft_Scan_Turntable_Axis.Position[1].Vel := 10000;
   PRODUCT_TYPE[4].Motion.Shaft_Scan_Turntable_Axis.Position[1].Pos := 0;
   PRODUCT_TYPE[4].Motion.Shaft_Scan_Turntable_Axis.Position[1].Vel := 10000;
   PRODUCT_TYPE[5].Motion.Shaft_Scan_Turntable_Axis.Position[1].Pos := 0;
   PRODUCT_TYPE[5].Motion.Shaft_Scan_Turntable_Axis.Position[1].Vel := 10000;
   PRODUCT_TYPE[6].Motion.Shaft_Scan_Turntable_Axis.Position[1].Pos := 0;
   PRODUCT_TYPE[6].Motion.Shaft_Scan_Turntable_Axis.Position[1].Vel := 10000;
   PRODUCT_TYPE[7].Motion.Shaft_Scan_Turntable_Axis.Position[1].Pos := 0;
   PRODUCT_TYPE[7].Motion.Shaft_Scan_Turntable_Axis.Position[1].Vel := 10000;
   PRODUCT_TYPE[8].Motion.Shaft_Scan_Turntable_Axis.Position[1].Pos := 0;
   PRODUCT_TYPE[8].Motion.Shaft_Scan_Turntable_Axis.Position[1].Vel := 10000;
   PRODUCT_TYPE[9].Motion.Shaft_Scan_Turntable_Axis.Position[1].Pos := 0;
   PRODUCT_TYPE[9].Motion.Shaft_Scan_Turntable_Axis.Position[1].Vel := 10000;
   PRODUCT_TYPE[10].Motion.Shaft_Scan_Turntable_Axis.Position[1].Pos := 0;
   PRODUCT_TYPE[10].Motion.Shaft_Scan_Turntable_Axis.Position[1].Vel := 10000;
   PRODUCT_TYPE[1].Motion.Shaft_Scan_Turntable_Axis.Position[2].Pos := 450000;
   PRODUCT_TYPE[1].Motion.Shaft_Scan_Turntable_Axis.Position[2].Vel := 10000;
   PRODUCT_TYPE[2].Motion.Shaft_Scan_Turntable_Axis.Position[2].Pos := 450000;
   PRODUCT_TYPE[2].Motion.Shaft_Scan_Turntable_Axis.Position[2].Vel := 10000;
   PRODUCT_TYPE[3].Motion.Shaft_Scan_Turntable_Axis.Position[2].Pos := 450000;
   PRODUCT_TYPE[3].Motion.Shaft_Scan_Turntable_Axis.Position[2].Vel := 10000;
   PRODUCT_TYPE[4].Motion.Shaft_Scan_Turntable_Axis.Position[2].Pos := 450000;
   PRODUCT_TYPE[4].Motion.Shaft_Scan_Turntable_Axis.Position[2].Vel := 10000;
   PRODUCT_TYPE[5].Motion.Shaft_Scan_Turntable_Axis.Position[2].Pos := 450000;
   PRODUCT_TYPE[5].Motion.Shaft_Scan_Turntable_Axis.Position[2].Vel := 10000;
   PRODUCT_TYPE[6].Motion.Shaft_Scan_Turntable_Axis.Position[2].Pos := 450000;
   PRODUCT_TYPE[6].Motion.Shaft_Scan_Turntable_Axis.Position[2].Vel := 10000;
   PRODUCT_TYPE[7].Motion.Shaft_Scan_Turntable_Axis.Position[2].Pos := 450000;
   PRODUCT_TYPE[7].Motion.Shaft_Scan_Turntable_Axis.Position[2].Vel := 10000;
   PRODUCT_TYPE[8].Motion.Shaft_Scan_Turntable_Axis.Position[2].Pos := 450000;
   PRODUCT_TYPE[8].Motion.Shaft_Scan_Turntable_Axis.Position[2].Vel := 10000;
   PRODUCT_TYPE[9].Motion.Shaft_Scan_Turntable_Axis.Position[2].Pos := 450000;
   PRODUCT_TYPE[9].Motion.Shaft_Scan_Turntable_Axis.Position[2].Vel := 10000;
   PRODUCT_TYPE[10].Motion.Shaft_Scan_Turntable_Axis.Position[2].Pos := 450000;
   PRODUCT_TYPE[10].Motion.Shaft_Scan_Turntable_Axis.Position[2].Vel := 10000;
   PRODUCT_TYPE[1].Motion.Shaft_Scan_Turntable_Axis.Position[3].Pos := 900000;
   PRODUCT_TYPE[1].Motion.Shaft_Scan_Turntable_Axis.Position[3].Vel := 10000;
   PRODUCT_TYPE[2].Motion.Shaft_Scan_Turntable_Axis.Position[3].Pos := 900000;
   PRODUCT_TYPE[2].Motion.Shaft_Scan_Turntable_Axis.Position[3].Vel := 10000;
   PRODUCT_TYPE[3].Motion.Shaft_Scan_Turntable_Axis.Position[3].Pos := 900000;
   PRODUCT_TYPE[3].Motion.Shaft_Scan_Turntable_Axis.Position[3].Vel := 10000;
   PRODUCT_TYPE[4].Motion.Shaft_Scan_Turntable_Axis.Position[3].Pos := 900000;
   PRODUCT_TYPE[4].Motion.Shaft_Scan_Turntable_Axis.Position[3].Vel := 10000;
   PRODUCT_TYPE[5].Motion.Shaft_Scan_Turntable_Axis.Position[3].Pos := 900000;
   PRODUCT_TYPE[5].Motion.Shaft_Scan_Turntable_Axis.Position[3].Vel := 10000;
   PRODUCT_TYPE[6].Motion.Shaft_Scan_Turntable_Axis.Position[3].Pos := 900000;
   PRODUCT_TYPE[6].Motion.Shaft_Scan_Turntable_Axis.Position[3].Vel := 10000;
   PRODUCT_TYPE[7].Motion.Shaft_Scan_Turntable_Axis.Position[3].Pos := 900000;
   PRODUCT_TYPE[7].Motion.Shaft_Scan_Turntable_Axis.Position[3].Vel := 10000;
   PRODUCT_TYPE[8].Motion.Shaft_Scan_Turntable_Axis.Position[3].Pos := 900000;
   PRODUCT_TYPE[8].Motion.Shaft_Scan_Turntable_Axis.Position[3].Vel := 10000;
   PRODUCT_TYPE[9].Motion.Shaft_Scan_Turntable_Axis.Position[3].Pos := 900000;
   PRODUCT_TYPE[9].Motion.Shaft_Scan_Turntable_Axis.Position[3].Vel := 10000;
   PRODUCT_TYPE[10].Motion.Shaft_Scan_Turntable_Axis.Position[3].Pos := 900000;
   PRODUCT_TYPE[10].Motion.Shaft_Scan_Turntable_Axis.Position[3].Vel := 10000;
   PRODUCT_TYPE[1].Motion.Shaft_Scan_Turntable_Axis.Position[4].Pos := 135000;
   PRODUCT_TYPE[1].Motion.Shaft_Scan_Turntable_Axis.Position[4].Vel := 10000;
   PRODUCT_TYPE[2].Motion.Shaft_Scan_Turntable_Axis.Position[4].Pos := 135000;
   PRODUCT_TYPE[2].Motion.Shaft_Scan_Turntable_Axis.Position[4].Vel := 10000;
   PRODUCT_TYPE[3].Motion.Shaft_Scan_Turntable_Axis.Position[4].Pos := 135000;
   PRODUCT_TYPE[3].Motion.Shaft_Scan_Turntable_Axis.Position[4].Vel := 10000;
   PRODUCT_TYPE[4].Motion.Shaft_Scan_Turntable_Axis.Position[4].Pos := 135000;
   PRODUCT_TYPE[4].Motion.Shaft_Scan_Turntable_Axis.Position[4].Vel := 10000;
   PRODUCT_TYPE[5].Motion.Shaft_Scan_Turntable_Axis.Position[4].Pos := 135000;
   PRODUCT_TYPE[5].Motion.Shaft_Scan_Turntable_Axis.Position[4].Vel := 10000;
   PRODUCT_TYPE[6].Motion.Shaft_Scan_Turntable_Axis.Position[4].Pos := 135000;
   PRODUCT_TYPE[6].Motion.Shaft_Scan_Turntable_Axis.Position[4].Vel := 10000;
   PRODUCT_TYPE[7].Motion.Shaft_Scan_Turntable_Axis.Position[4].Pos := 135000;
   PRODUCT_TYPE[7].Motion.Shaft_Scan_Turntable_Axis.Position[4].Vel := 10000;
   PRODUCT_TYPE[8].Motion.Shaft_Scan_Turntable_Axis.Position[4].Pos := 135000;
   PRODUCT_TYPE[8].Motion.Shaft_Scan_Turntable_Axis.Position[4].Vel := 10000;
   PRODUCT_TYPE[9].Motion.Shaft_Scan_Turntable_Axis.Position[4].Pos := 135000;
   PRODUCT_TYPE[9].Motion.Shaft_Scan_Turntable_Axis.Position[4].Vel := 10000;
   PRODUCT_TYPE[10].Motion.Shaft_Scan_Turntable_Axis.Position[4].Pos := 135000;
   PRODUCT_TYPE[10].Motion.Shaft_Scan_Turntable_Axis.Position[4].Vel := 10000;
   PRODUCT_TYPE[1].Motion.Shaft_Scan_Turntable_Axis.Position[5].Pos := 180000;
   PRODUCT_TYPE[1].Motion.Shaft_Scan_Turntable_Axis.Position[5].Vel := 10000;
   PRODUCT_TYPE[2].Motion.Shaft_Scan_Turntable_Axis.Position[5].Pos := 180000;
   PRODUCT_TYPE[2].Motion.Shaft_Scan_Turntable_Axis.Position[5].Vel := 10000;
   PRODUCT_TYPE[3].Motion.Shaft_Scan_Turntable_Axis.Position[5].Pos := 180000;
   PRODUCT_TYPE[3].Motion.Shaft_Scan_Turntable_Axis.Position[5].Vel := 10000;
   PRODUCT_TYPE[4].Motion.Shaft_Scan_Turntable_Axis.Position[5].Pos := 180000;
   PRODUCT_TYPE[4].Motion.Shaft_Scan_Turntable_Axis.Position[5].Vel := 10000;
   PRODUCT_TYPE[5].Motion.Shaft_Scan_Turntable_Axis.Position[5].Pos := 180000;
   PRODUCT_TYPE[5].Motion.Shaft_Scan_Turntable_Axis.Position[5].Vel := 10000;
   PRODUCT_TYPE[6].Motion.Shaft_Scan_Turntable_Axis.Position[5].Pos := 180000;
   PRODUCT_TYPE[6].Motion.Shaft_Scan_Turntable_Axis.Position[5].Vel := 10000;
   PRODUCT_TYPE[7].Motion.Shaft_Scan_Turntable_Axis.Position[5].Pos := 180000;
   PRODUCT_TYPE[7].Motion.Shaft_Scan_Turntable_Axis.Position[5].Vel := 10000;
   PRODUCT_TYPE[8].Motion.Shaft_Scan_Turntable_Axis.Position[5].Pos := 180000;
   PRODUCT_TYPE[8].Motion.Shaft_Scan_Turntable_Axis.Position[5].Vel := 10000;
   PRODUCT_TYPE[9].Motion.Shaft_Scan_Turntable_Axis.Position[5].Pos := 180000;
   PRODUCT_TYPE[9].Motion.Shaft_Scan_Turntable_Axis.Position[5].Vel := 10000;
   PRODUCT_TYPE[10].Motion.Shaft_Scan_Turntable_Axis.Position[5].Pos := 180000;
   PRODUCT_TYPE[10].Motion.Shaft_Scan_Turntable_Axis.Position[5].Vel := 10000;
   PRODUCT_TYPE[1].Motion.Shaft_Scan_Turntable_Axis.Position[6].Pos := 225000;
   PRODUCT_TYPE[1].Motion.Shaft_Scan_Turntable_Axis.Position[6].Vel := 10000;
   PRODUCT_TYPE[2].Motion.Shaft_Scan_Turntable_Axis.Position[6].Pos := 225000;
   PRODUCT_TYPE[2].Motion.Shaft_Scan_Turntable_Axis.Position[6].Vel := 10000;
   PRODUCT_TYPE[3].Motion.Shaft_Scan_Turntable_Axis.Position[6].Pos := 225000;
   PRODUCT_TYPE[3].Motion.Shaft_Scan_Turntable_Axis.Position[6].Vel := 10000;
   PRODUCT_TYPE[4].Motion.Shaft_Scan_Turntable_Axis.Position[6].Pos := 225000;
   PRODUCT_TYPE[4].Motion.Shaft_Scan_Turntable_Axis.Position[6].Vel := 10000;
   PRODUCT_TYPE[5].Motion.Shaft_Scan_Turntable_Axis.Position[6].Pos := 225000;
   PRODUCT_TYPE[5].Motion.Shaft_Scan_Turntable_Axis.Position[6].Vel := 10000;
   PRODUCT_TYPE[6].Motion.Shaft_Scan_Turntable_Axis.Position[6].Pos := 225000;
   PRODUCT_TYPE[6].Motion.Shaft_Scan_Turntable_Axis.Position[6].Vel := 10000;
   PRODUCT_TYPE[7].Motion.Shaft_Scan_Turntable_Axis.Position[6].Pos := 225000;
   PRODUCT_TYPE[7].Motion.Shaft_Scan_Turntable_Axis.Position[6].Vel := 10000;
   PRODUCT_TYPE[8].Motion.Shaft_Scan_Turntable_Axis.Position[6].Pos := 225000;
   PRODUCT_TYPE[8].Motion.Shaft_Scan_Turntable_Axis.Position[6].Vel := 10000;
   PRODUCT_TYPE[9].Motion.Shaft_Scan_Turntable_Axis.Position[6].Pos := 225000;
   PRODUCT_TYPE[9].Motion.Shaft_Scan_Turntable_Axis.Position[6].Vel := 10000;
   PRODUCT_TYPE[10].Motion.Shaft_Scan_Turntable_Axis.Position[6].Pos := 225000;
   PRODUCT_TYPE[10].Motion.Shaft_Scan_Turntable_Axis.Position[6].Vel := 10000;
   PRODUCT_TYPE[1].Motion.Shaft_Scan_Turntable_Axis.Position[7].Pos := 270000;
   PRODUCT_TYPE[1].Motion.Shaft_Scan_Turntable_Axis.Position[7].Vel := 10000;
   PRODUCT_TYPE[2].Motion.Shaft_Scan_Turntable_Axis.Position[7].Pos := 270000;
   PRODUCT_TYPE[2].Motion.Shaft_Scan_Turntable_Axis.Position[7].Vel := 10000;
   PRODUCT_TYPE[3].Motion.Shaft_Scan_Turntable_Axis.Position[7].Pos := 270000;
   PRODUCT_TYPE[3].Motion.Shaft_Scan_Turntable_Axis.Position[7].Vel := 10000;
   PRODUCT_TYPE[4].Motion.Shaft_Scan_Turntable_Axis.Position[7].Pos := 270000;
   PRODUCT_TYPE[4].Motion.Shaft_Scan_Turntable_Axis.Position[7].Vel := 10000;
   PRODUCT_TYPE[5].Motion.Shaft_Scan_Turntable_Axis.Position[7].Pos := 270000;
   PRODUCT_TYPE[5].Motion.Shaft_Scan_Turntable_Axis.Position[7].Vel := 10000;
   PRODUCT_TYPE[6].Motion.Shaft_Scan_Turntable_Axis.Position[7].Pos := 270000;
   PRODUCT_TYPE[6].Motion.Shaft_Scan_Turntable_Axis.Position[7].Vel := 10000;
   PRODUCT_TYPE[7].Motion.Shaft_Scan_Turntable_Axis.Position[7].Pos := 270000;
   PRODUCT_TYPE[7].Motion.Shaft_Scan_Turntable_Axis.Position[7].Vel := 10000;
   PRODUCT_TYPE[8].Motion.Shaft_Scan_Turntable_Axis.Position[7].Pos := 270000;
   PRODUCT_TYPE[8].Motion.Shaft_Scan_Turntable_Axis.Position[7].Vel := 10000;
   PRODUCT_TYPE[9].Motion.Shaft_Scan_Turntable_Axis.Position[7].Pos := 270000;
   PRODUCT_TYPE[9].Motion.Shaft_Scan_Turntable_Axis.Position[7].Vel := 10000;
   PRODUCT_TYPE[10].Motion.Shaft_Scan_Turntable_Axis.Position[7].Pos := 270000;
   PRODUCT_TYPE[10].Motion.Shaft_Scan_Turntable_Axis.Position[7].Vel := 10000;
   PRODUCT_TYPE[1].Motion.Shaft_Scan_Turntable_Axis.Position[8].Pos := 315000;
   PRODUCT_TYPE[1].Motion.Shaft_Scan_Turntable_Axis.Position[8].Vel := 10000;
   PRODUCT_TYPE[2].Motion.Shaft_Scan_Turntable_Axis.Position[8].Pos := 315000;
   PRODUCT_TYPE[2].Motion.Shaft_Scan_Turntable_Axis.Position[8].Vel := 10000;
   PRODUCT_TYPE[3].Motion.Shaft_Scan_Turntable_Axis.Position[8].Pos := 315000;
   PRODUCT_TYPE[3].Motion.Shaft_Scan_Turntable_Axis.Position[8].Vel := 10000;
   PRODUCT_TYPE[4].Motion.Shaft_Scan_Turntable_Axis.Position[8].Pos := 315000;
   PRODUCT_TYPE[4].Motion.Shaft_Scan_Turntable_Axis.Position[8].Vel := 10000;
   PRODUCT_TYPE[5].Motion.Shaft_Scan_Turntable_Axis.Position[8].Pos := 315000;
   PRODUCT_TYPE[5].Motion.Shaft_Scan_Turntable_Axis.Position[8].Vel := 10000;
   PRODUCT_TYPE[6].Motion.Shaft_Scan_Turntable_Axis.Position[8].Pos := 315000;
   PRODUCT_TYPE[6].Motion.Shaft_Scan_Turntable_Axis.Position[8].Vel := 10000;
   PRODUCT_TYPE[7].Motion.Shaft_Scan_Turntable_Axis.Position[8].Pos := 315000;
   PRODUCT_TYPE[7].Motion.Shaft_Scan_Turntable_Axis.Position[8].Vel := 10000;
   PRODUCT_TYPE[8].Motion.Shaft_Scan_Turntable_Axis.Position[8].Pos := 315000;
   PRODUCT_TYPE[8].Motion.Shaft_Scan_Turntable_Axis.Position[8].Vel := 10000;
   PRODUCT_TYPE[9].Motion.Shaft_Scan_Turntable_Axis.Position[8].Pos := 315000;
   PRODUCT_TYPE[9].Motion.Shaft_Scan_Turntable_Axis.Position[8].Vel := 10000;
   PRODUCT_TYPE[10].Motion.Shaft_Scan_Turntable_Axis.Position[8].Pos := 315000;
   PRODUCT_TYPE[10].Motion.Shaft_Scan_Turntable_Axis.Position[8].Vel := 10000;
   PRODUCT_TYPE[1].Motion.Shaft_Scan_Turntable_Axis.Position[9].Pos := 0;
   PRODUCT_TYPE[1].Motion.Shaft_Scan_Turntable_Axis.Position[9].Vel := 0;
   PRODUCT_TYPE[2].Motion.Shaft_Scan_Turntable_Axis.Position[9].Pos := 0;
   PRODUCT_TYPE[2].Motion.Shaft_Scan_Turntable_Axis.Position[9].Vel := 0;
   PRODUCT_TYPE[3].Motion.Shaft_Scan_Turntable_Axis.Position[9].Pos := 0;
   PRODUCT_TYPE[3].Motion.Shaft_Scan_Turntable_Axis.Position[9].Vel := 0;
   PRODUCT_TYPE[4].Motion.Shaft_Scan_Turntable_Axis.Position[9].Pos := 0;
   PRODUCT_TYPE[4].Motion.Shaft_Scan_Turntable_Axis.Position[9].Vel := 0;
   PRODUCT_TYPE[5].Motion.Shaft_Scan_Turntable_Axis.Position[9].Pos := 0;
   PRODUCT_TYPE[5].Motion.Shaft_Scan_Turntable_Axis.Position[9].Vel := 0;
   PRODUCT_TYPE[6].Motion.Shaft_Scan_Turntable_Axis.Position[9].Pos := 0;
   PRODUCT_TYPE[6].Motion.Shaft_Scan_Turntable_Axis.Position[9].Vel := 0;
   PRODUCT_TYPE[7].Motion.Shaft_Scan_Turntable_Axis.Position[9].Pos := 0;
   PRODUCT_TYPE[7].Motion.Shaft_Scan_Turntable_Axis.Position[9].Vel := 0;
   PRODUCT_TYPE[8].Motion.Shaft_Scan_Turntable_Axis.Position[9].Pos := 0;
   PRODUCT_TYPE[8].Motion.Shaft_Scan_Turntable_Axis.Position[9].Vel := 0;
   PRODUCT_TYPE[9].Motion.Shaft_Scan_Turntable_Axis.Position[9].Pos := 0;
   PRODUCT_TYPE[9].Motion.Shaft_Scan_Turntable_Axis.Position[9].Vel := 0;
   PRODUCT_TYPE[10].Motion.Shaft_Scan_Turntable_Axis.Position[9].Pos := 0;
   PRODUCT_TYPE[10].Motion.Shaft_Scan_Turntable_Axis.Position[9].Vel := 0;
   PRODUCT_TYPE[1].Motion.Shaft_Scan_Turntable_Axis.Position[10].Pos := 0;
   PRODUCT_TYPE[1].Motion.Shaft_Scan_Turntable_Axis.Position[10].Vel := 0;
   PRODUCT_TYPE[2].Motion.Shaft_Scan_Turntable_Axis.Position[10].Pos := 0;
   PRODUCT_TYPE[2].Motion.Shaft_Scan_Turntable_Axis.Position[10].Vel := 0;
   PRODUCT_TYPE[3].Motion.Shaft_Scan_Turntable_Axis.Position[10].Pos := 0;
   PRODUCT_TYPE[3].Motion.Shaft_Scan_Turntable_Axis.Position[10].Vel := 0;
   PRODUCT_TYPE[4].Motion.Shaft_Scan_Turntable_Axis.Position[10].Pos := 0;
   PRODUCT_TYPE[4].Motion.Shaft_Scan_Turntable_Axis.Position[10].Vel := 0;
   PRODUCT_TYPE[5].Motion.Shaft_Scan_Turntable_Axis.Position[10].Pos := 0;
   PRODUCT_TYPE[5].Motion.Shaft_Scan_Turntable_Axis.Position[10].Vel := 0;
   PRODUCT_TYPE[6].Motion.Shaft_Scan_Turntable_Axis.Position[10].Pos := 0;
   PRODUCT_TYPE[6].Motion.Shaft_Scan_Turntable_Axis.Position[10].Vel := 0;
   PRODUCT_TYPE[7].Motion.Shaft_Scan_Turntable_Axis.Position[10].Pos := 0;
   PRODUCT_TYPE[7].Motion.Shaft_Scan_Turntable_Axis.Position[10].Vel := 0;
   PRODUCT_TYPE[8].Motion.Shaft_Scan_Turntable_Axis.Position[10].Pos := 0;
   PRODUCT_TYPE[8].Motion.Shaft_Scan_Turntable_Axis.Position[10].Vel := 0;
   PRODUCT_TYPE[9].Motion.Shaft_Scan_Turntable_Axis.Position[10].Pos := 0;
   PRODUCT_TYPE[9].Motion.Shaft_Scan_Turntable_Axis.Position[10].Vel := 0;
   PRODUCT_TYPE[10].Motion.Shaft_Scan_Turntable_Axis.Position[10].Pos := 0;
   PRODUCT_TYPE[10].Motion.Shaft_Scan_Turntable_Axis.Position[10].Vel := 0;
   PRODUCT_TYPE[1].Motion.Shaft_Scan_Turntable_Axis.Position[11].Pos := 0;
   PRODUCT_TYPE[1].Motion.Shaft_Scan_Turntable_Axis.Position[11].Vel := 0;
   PRODUCT_TYPE[2].Motion.Shaft_Scan_Turntable_Axis.Position[11].Pos := 0;
   PRODUCT_TYPE[2].Motion.Shaft_Scan_Turntable_Axis.Position[11].Vel := 0;
   PRODUCT_TYPE[3].Motion.Shaft_Scan_Turntable_Axis.Position[11].Pos := 0;
   PRODUCT_TYPE[3].Motion.Shaft_Scan_Turntable_Axis.Position[11].Vel := 0;
   PRODUCT_TYPE[4].Motion.Shaft_Scan_Turntable_Axis.Position[11].Pos := 0;
   PRODUCT_TYPE[4].Motion.Shaft_Scan_Turntable_Axis.Position[11].Vel := 0;
   PRODUCT_TYPE[5].Motion.Shaft_Scan_Turntable_Axis.Position[11].Pos := 0;
   PRODUCT_TYPE[5].Motion.Shaft_Scan_Turntable_Axis.Position[11].Vel := 0;
   PRODUCT_TYPE[6].Motion.Shaft_Scan_Turntable_Axis.Position[11].Pos := 0;
   PRODUCT_TYPE[6].Motion.Shaft_Scan_Turntable_Axis.Position[11].Vel := 0;
   PRODUCT_TYPE[7].Motion.Shaft_Scan_Turntable_Axis.Position[11].Pos := 0;
   PRODUCT_TYPE[7].Motion.Shaft_Scan_Turntable_Axis.Position[11].Vel := 0;
   PRODUCT_TYPE[8].Motion.Shaft_Scan_Turntable_Axis.Position[11].Pos := 0;
   PRODUCT_TYPE[8].Motion.Shaft_Scan_Turntable_Axis.Position[11].Vel := 0;
   PRODUCT_TYPE[9].Motion.Shaft_Scan_Turntable_Axis.Position[11].Pos := 0;
   PRODUCT_TYPE[9].Motion.Shaft_Scan_Turntable_Axis.Position[11].Vel := 0;
   PRODUCT_TYPE[10].Motion.Shaft_Scan_Turntable_Axis.Position[11].Pos := 0;
   PRODUCT_TYPE[10].Motion.Shaft_Scan_Turntable_Axis.Position[11].Vel := 0;
   PRODUCT_TYPE[1].Motion.Shaft_Scan_Turntable_Axis.Position[12].Pos := 0;
   PRODUCT_TYPE[1].Motion.Shaft_Scan_Turntable_Axis.Position[12].Vel := 0;
   PRODUCT_TYPE[2].Motion.Shaft_Scan_Turntable_Axis.Position[12].Pos := 0;
   PRODUCT_TYPE[2].Motion.Shaft_Scan_Turntable_Axis.Position[12].Vel := 0;
   PRODUCT_TYPE[3].Motion.Shaft_Scan_Turntable_Axis.Position[12].Pos := 0;
   PRODUCT_TYPE[3].Motion.Shaft_Scan_Turntable_Axis.Position[12].Vel := 0;
   PRODUCT_TYPE[4].Motion.Shaft_Scan_Turntable_Axis.Position[12].Pos := 0;
   PRODUCT_TYPE[4].Motion.Shaft_Scan_Turntable_Axis.Position[12].Vel := 0;
   PRODUCT_TYPE[5].Motion.Shaft_Scan_Turntable_Axis.Position[12].Pos := 0;
   PRODUCT_TYPE[5].Motion.Shaft_Scan_Turntable_Axis.Position[12].Vel := 0;
   PRODUCT_TYPE[6].Motion.Shaft_Scan_Turntable_Axis.Position[12].Pos := 0;
   PRODUCT_TYPE[6].Motion.Shaft_Scan_Turntable_Axis.Position[12].Vel := 0;
   PRODUCT_TYPE[7].Motion.Shaft_Scan_Turntable_Axis.Position[12].Pos := 0;
   PRODUCT_TYPE[7].Motion.Shaft_Scan_Turntable_Axis.Position[12].Vel := 0;
   PRODUCT_TYPE[8].Motion.Shaft_Scan_Turntable_Axis.Position[12].Pos := 0;
   PRODUCT_TYPE[8].Motion.Shaft_Scan_Turntable_Axis.Position[12].Vel := 0;
   PRODUCT_TYPE[9].Motion.Shaft_Scan_Turntable_Axis.Position[12].Pos := 0;
   PRODUCT_TYPE[9].Motion.Shaft_Scan_Turntable_Axis.Position[12].Vel := 0;
   PRODUCT_TYPE[10].Motion.Shaft_Scan_Turntable_Axis.Position[12].Pos := 0;
   PRODUCT_TYPE[10].Motion.Shaft_Scan_Turntable_Axis.Position[12].Vel := 0;
   PRODUCT_TYPE[1].Motion.Shaft_Scan_Turntable_Axis.Position[13].Pos := 0;
   PRODUCT_TYPE[1].Motion.Shaft_Scan_Turntable_Axis.Position[13].Vel := 0;
   PRODUCT_TYPE[2].Motion.Shaft_Scan_Turntable_Axis.Position[13].Pos := 0;
   PRODUCT_TYPE[2].Motion.Shaft_Scan_Turntable_Axis.Position[13].Vel := 0;
   PRODUCT_TYPE[3].Motion.Shaft_Scan_Turntable_Axis.Position[13].Pos := 0;
   PRODUCT_TYPE[3].Motion.Shaft_Scan_Turntable_Axis.Position[13].Vel := 0;
   PRODUCT_TYPE[4].Motion.Shaft_Scan_Turntable_Axis.Position[13].Pos := 0;
   PRODUCT_TYPE[4].Motion.Shaft_Scan_Turntable_Axis.Position[13].Vel := 0;
   PRODUCT_TYPE[5].Motion.Shaft_Scan_Turntable_Axis.Position[13].Pos := 0;
   PRODUCT_TYPE[5].Motion.Shaft_Scan_Turntable_Axis.Position[13].Vel := 0;
   PRODUCT_TYPE[6].Motion.Shaft_Scan_Turntable_Axis.Position[13].Pos := 0;
   PRODUCT_TYPE[6].Motion.Shaft_Scan_Turntable_Axis.Position[13].Vel := 0;
   PRODUCT_TYPE[7].Motion.Shaft_Scan_Turntable_Axis.Position[13].Pos := 0;
   PRODUCT_TYPE[7].Motion.Shaft_Scan_Turntable_Axis.Position[13].Vel := 0;
   PRODUCT_TYPE[8].Motion.Shaft_Scan_Turntable_Axis.Position[13].Pos := 0;
   PRODUCT_TYPE[8].Motion.Shaft_Scan_Turntable_Axis.Position[13].Vel := 0;
   PRODUCT_TYPE[9].Motion.Shaft_Scan_Turntable_Axis.Position[13].Pos := 0;
   PRODUCT_TYPE[9].Motion.Shaft_Scan_Turntable_Axis.Position[13].Vel := 0;
   PRODUCT_TYPE[10].Motion.Shaft_Scan_Turntable_Axis.Position[13].Pos := 0;
   PRODUCT_TYPE[10].Motion.Shaft_Scan_Turntable_Axis.Position[13].Vel := 0;
   PRODUCT_TYPE[1].Motion.Shaft_Scan_Turntable_Axis.Position[14].Pos := 0;
   PRODUCT_TYPE[1].Motion.Shaft_Scan_Turntable_Axis.Position[14].Vel := 0;
   PRODUCT_TYPE[2].Motion.Shaft_Scan_Turntable_Axis.Position[14].Pos := 0;
   PRODUCT_TYPE[2].Motion.Shaft_Scan_Turntable_Axis.Position[14].Vel := 0;
   PRODUCT_TYPE[3].Motion.Shaft_Scan_Turntable_Axis.Position[14].Pos := 0;
   PRODUCT_TYPE[3].Motion.Shaft_Scan_Turntable_Axis.Position[14].Vel := 0;
   PRODUCT_TYPE[4].Motion.Shaft_Scan_Turntable_Axis.Position[14].Pos := 0;
   PRODUCT_TYPE[4].Motion.Shaft_Scan_Turntable_Axis.Position[14].Vel := 0;
   PRODUCT_TYPE[5].Motion.Shaft_Scan_Turntable_Axis.Position[14].Pos := 0;
   PRODUCT_TYPE[5].Motion.Shaft_Scan_Turntable_Axis.Position[14].Vel := 0;
   PRODUCT_TYPE[6].Motion.Shaft_Scan_Turntable_Axis.Position[14].Pos := 0;
   PRODUCT_TYPE[6].Motion.Shaft_Scan_Turntable_Axis.Position[14].Vel := 0;
   PRODUCT_TYPE[7].Motion.Shaft_Scan_Turntable_Axis.Position[14].Pos := 0;
   PRODUCT_TYPE[7].Motion.Shaft_Scan_Turntable_Axis.Position[14].Vel := 0;
   PRODUCT_TYPE[8].Motion.Shaft_Scan_Turntable_Axis.Position[14].Pos := 0;
   PRODUCT_TYPE[8].Motion.Shaft_Scan_Turntable_Axis.Position[14].Vel := 0;
   PRODUCT_TYPE[9].Motion.Shaft_Scan_Turntable_Axis.Position[14].Pos := 0;
   PRODUCT_TYPE[9].Motion.Shaft_Scan_Turntable_Axis.Position[14].Vel := 0;
   PRODUCT_TYPE[10].Motion.Shaft_Scan_Turntable_Axis.Position[14].Pos := 0;
   PRODUCT_TYPE[10].Motion.Shaft_Scan_Turntable_Axis.Position[14].Vel := 0;
   PRODUCT_TYPE[1].Motion.Shaft_Scan_Turntable_Axis.Position[15].Pos := 0;
   PRODUCT_TYPE[1].Motion.Shaft_Scan_Turntable_Axis.Position[15].Vel := 0;
   PRODUCT_TYPE[2].Motion.Shaft_Scan_Turntable_Axis.Position[15].Pos := 0;
   PRODUCT_TYPE[2].Motion.Shaft_Scan_Turntable_Axis.Position[15].Vel := 0;
   PRODUCT_TYPE[3].Motion.Shaft_Scan_Turntable_Axis.Position[15].Pos := 0;
   PRODUCT_TYPE[3].Motion.Shaft_Scan_Turntable_Axis.Position[15].Vel := 0;
   PRODUCT_TYPE[4].Motion.Shaft_Scan_Turntable_Axis.Position[15].Pos := 0;
   PRODUCT_TYPE[4].Motion.Shaft_Scan_Turntable_Axis.Position[15].Vel := 0;
   PRODUCT_TYPE[5].Motion.Shaft_Scan_Turntable_Axis.Position[15].Pos := 0;
   PRODUCT_TYPE[5].Motion.Shaft_Scan_Turntable_Axis.Position[15].Vel := 0;
   PRODUCT_TYPE[6].Motion.Shaft_Scan_Turntable_Axis.Position[15].Pos := 0;
   PRODUCT_TYPE[6].Motion.Shaft_Scan_Turntable_Axis.Position[15].Vel := 0;
   PRODUCT_TYPE[7].Motion.Shaft_Scan_Turntable_Axis.Position[15].Pos := 0;
   PRODUCT_TYPE[7].Motion.Shaft_Scan_Turntable_Axis.Position[15].Vel := 0;
   PRODUCT_TYPE[8].Motion.Shaft_Scan_Turntable_Axis.Position[15].Pos := 0;
   PRODUCT_TYPE[8].Motion.Shaft_Scan_Turntable_Axis.Position[15].Vel := 0;
   PRODUCT_TYPE[9].Motion.Shaft_Scan_Turntable_Axis.Position[15].Pos := 0;
   PRODUCT_TYPE[9].Motion.Shaft_Scan_Turntable_Axis.Position[15].Vel := 0;
   PRODUCT_TYPE[10].Motion.Shaft_Scan_Turntable_Axis.Position[15].Pos := 0;
   PRODUCT_TYPE[10].Motion.Shaft_Scan_Turntable_Axis.Position[15].Vel := 0;
   PRODUCT_TYPE[1].Motion.Shaft_Scan_Turntable_Axis.Position[16].Pos := 0;
   PRODUCT_TYPE[1].Motion.Shaft_Scan_Turntable_Axis.Position[16].Vel := 0;
   PRODUCT_TYPE[2].Motion.Shaft_Scan_Turntable_Axis.Position[16].Pos := 0;
   PRODUCT_TYPE[2].Motion.Shaft_Scan_Turntable_Axis.Position[16].Vel := 0;
   PRODUCT_TYPE[3].Motion.Shaft_Scan_Turntable_Axis.Position[16].Pos := 0;
   PRODUCT_TYPE[3].Motion.Shaft_Scan_Turntable_Axis.Position[16].Vel := 0;
   PRODUCT_TYPE[4].Motion.Shaft_Scan_Turntable_Axis.Position[16].Pos := 0;
   PRODUCT_TYPE[4].Motion.Shaft_Scan_Turntable_Axis.Position[16].Vel := 0;
   PRODUCT_TYPE[5].Motion.Shaft_Scan_Turntable_Axis.Position[16].Pos := 0;
   PRODUCT_TYPE[5].Motion.Shaft_Scan_Turntable_Axis.Position[16].Vel := 0;
   PRODUCT_TYPE[6].Motion.Shaft_Scan_Turntable_Axis.Position[16].Pos := 0;
   PRODUCT_TYPE[6].Motion.Shaft_Scan_Turntable_Axis.Position[16].Vel := 0;
   PRODUCT_TYPE[7].Motion.Shaft_Scan_Turntable_Axis.Position[16].Pos := 0;
   PRODUCT_TYPE[7].Motion.Shaft_Scan_Turntable_Axis.Position[16].Vel := 0;
   PRODUCT_TYPE[8].Motion.Shaft_Scan_Turntable_Axis.Position[16].Pos := 0;
   PRODUCT_TYPE[8].Motion.Shaft_Scan_Turntable_Axis.Position[16].Vel := 0;
   PRODUCT_TYPE[9].Motion.Shaft_Scan_Turntable_Axis.Position[16].Pos := 0;
   PRODUCT_TYPE[9].Motion.Shaft_Scan_Turntable_Axis.Position[16].Vel := 0;
   PRODUCT_TYPE[10].Motion.Shaft_Scan_Turntable_Axis.Position[16].Pos := 0;
   PRODUCT_TYPE[10].Motion.Shaft_Scan_Turntable_Axis.Position[16].Vel := 0;
   PRODUCT_TYPE[1].Motion.Shaft_Scan_Turntable_Axis.Position[17].Pos := 0;
   PRODUCT_TYPE[1].Motion.Shaft_Scan_Turntable_Axis.Position[17].Vel := 0;
   PRODUCT_TYPE[2].Motion.Shaft_Scan_Turntable_Axis.Position[17].Pos := 0;
   PRODUCT_TYPE[2].Motion.Shaft_Scan_Turntable_Axis.Position[17].Vel := 0;
   PRODUCT_TYPE[3].Motion.Shaft_Scan_Turntable_Axis.Position[17].Pos := 0;
   PRODUCT_TYPE[3].Motion.Shaft_Scan_Turntable_Axis.Position[17].Vel := 0;
   PRODUCT_TYPE[4].Motion.Shaft_Scan_Turntable_Axis.Position[17].Pos := 0;
   PRODUCT_TYPE[4].Motion.Shaft_Scan_Turntable_Axis.Position[17].Vel := 0;
   PRODUCT_TYPE[5].Motion.Shaft_Scan_Turntable_Axis.Position[17].Pos := 0;
   PRODUCT_TYPE[5].Motion.Shaft_Scan_Turntable_Axis.Position[17].Vel := 0;
   PRODUCT_TYPE[6].Motion.Shaft_Scan_Turntable_Axis.Position[17].Pos := 0;
   PRODUCT_TYPE[6].Motion.Shaft_Scan_Turntable_Axis.Position[17].Vel := 0;
   PRODUCT_TYPE[7].Motion.Shaft_Scan_Turntable_Axis.Position[17].Pos := 0;
   PRODUCT_TYPE[7].Motion.Shaft_Scan_Turntable_Axis.Position[17].Vel := 0;
   PRODUCT_TYPE[8].Motion.Shaft_Scan_Turntable_Axis.Position[17].Pos := 0;
   PRODUCT_TYPE[8].Motion.Shaft_Scan_Turntable_Axis.Position[17].Vel := 0;
   PRODUCT_TYPE[9].Motion.Shaft_Scan_Turntable_Axis.Position[17].Pos := 0;
   PRODUCT_TYPE[9].Motion.Shaft_Scan_Turntable_Axis.Position[17].Vel := 0;
   PRODUCT_TYPE[10].Motion.Shaft_Scan_Turntable_Axis.Position[17].Pos := 0;
   PRODUCT_TYPE[10].Motion.Shaft_Scan_Turntable_Axis.Position[17].Vel := 0;
   PRODUCT_TYPE[1].Motion.Shaft_Scan_Turntable_Axis.Position[18].Pos := 0;
   PRODUCT_TYPE[1].Motion.Shaft_Scan_Turntable_Axis.Position[18].Vel := 0;
   PRODUCT_TYPE[2].Motion.Shaft_Scan_Turntable_Axis.Position[18].Pos := 0;
   PRODUCT_TYPE[2].Motion.Shaft_Scan_Turntable_Axis.Position[18].Vel := 0;
   PRODUCT_TYPE[3].Motion.Shaft_Scan_Turntable_Axis.Position[18].Pos := 0;
   PRODUCT_TYPE[3].Motion.Shaft_Scan_Turntable_Axis.Position[18].Vel := 0;
   PRODUCT_TYPE[4].Motion.Shaft_Scan_Turntable_Axis.Position[18].Pos := 0;
   PRODUCT_TYPE[4].Motion.Shaft_Scan_Turntable_Axis.Position[18].Vel := 0;
   PRODUCT_TYPE[5].Motion.Shaft_Scan_Turntable_Axis.Position[18].Pos := 0;
   PRODUCT_TYPE[5].Motion.Shaft_Scan_Turntable_Axis.Position[18].Vel := 0;
   PRODUCT_TYPE[6].Motion.Shaft_Scan_Turntable_Axis.Position[18].Pos := 0;
   PRODUCT_TYPE[6].Motion.Shaft_Scan_Turntable_Axis.Position[18].Vel := 0;
   PRODUCT_TYPE[7].Motion.Shaft_Scan_Turntable_Axis.Position[18].Pos := 0;
   PRODUCT_TYPE[7].Motion.Shaft_Scan_Turntable_Axis.Position[18].Vel := 0;
   PRODUCT_TYPE[8].Motion.Shaft_Scan_Turntable_Axis.Position[18].Pos := 0;
   PRODUCT_TYPE[8].Motion.Shaft_Scan_Turntable_Axis.Position[18].Vel := 0;
   PRODUCT_TYPE[9].Motion.Shaft_Scan_Turntable_Axis.Position[18].Pos := 0;
   PRODUCT_TYPE[9].Motion.Shaft_Scan_Turntable_Axis.Position[18].Vel := 0;
   PRODUCT_TYPE[10].Motion.Shaft_Scan_Turntable_Axis.Position[18].Pos := 0;
   PRODUCT_TYPE[10].Motion.Shaft_Scan_Turntable_Axis.Position[18].Vel := 0;
   PRODUCT_TYPE[1].Motion.Shaft_Scan_Turntable_Axis.Position[19].Pos := 0;
   PRODUCT_TYPE[1].Motion.Shaft_Scan_Turntable_Axis.Position[19].Vel := 0;
   PRODUCT_TYPE[2].Motion.Shaft_Scan_Turntable_Axis.Position[19].Pos := 0;
   PRODUCT_TYPE[2].Motion.Shaft_Scan_Turntable_Axis.Position[19].Vel := 0;
   PRODUCT_TYPE[3].Motion.Shaft_Scan_Turntable_Axis.Position[19].Pos := 0;
   PRODUCT_TYPE[3].Motion.Shaft_Scan_Turntable_Axis.Position[19].Vel := 0;
   PRODUCT_TYPE[4].Motion.Shaft_Scan_Turntable_Axis.Position[19].Pos := 0;
   PRODUCT_TYPE[4].Motion.Shaft_Scan_Turntable_Axis.Position[19].Vel := 0;
   PRODUCT_TYPE[5].Motion.Shaft_Scan_Turntable_Axis.Position[19].Pos := 0;
   PRODUCT_TYPE[5].Motion.Shaft_Scan_Turntable_Axis.Position[19].Vel := 0;
   PRODUCT_TYPE[6].Motion.Shaft_Scan_Turntable_Axis.Position[19].Pos := 0;
   PRODUCT_TYPE[6].Motion.Shaft_Scan_Turntable_Axis.Position[19].Vel := 0;
   PRODUCT_TYPE[7].Motion.Shaft_Scan_Turntable_Axis.Position[19].Pos := 0;
   PRODUCT_TYPE[7].Motion.Shaft_Scan_Turntable_Axis.Position[19].Vel := 0;
   PRODUCT_TYPE[8].Motion.Shaft_Scan_Turntable_Axis.Position[19].Pos := 0;
   PRODUCT_TYPE[8].Motion.Shaft_Scan_Turntable_Axis.Position[19].Vel := 0;
   PRODUCT_TYPE[9].Motion.Shaft_Scan_Turntable_Axis.Position[19].Pos := 0;
   PRODUCT_TYPE[9].Motion.Shaft_Scan_Turntable_Axis.Position[19].Vel := 0;
   PRODUCT_TYPE[10].Motion.Shaft_Scan_Turntable_Axis.Position[19].Pos := 0;
   PRODUCT_TYPE[10].Motion.Shaft_Scan_Turntable_Axis.Position[19].Vel := 0;
   PRODUCT_TYPE[1].Motion.Shaft_Scan_Turntable_Axis.Position[20].Pos := 0;
   PRODUCT_TYPE[1].Motion.Shaft_Scan_Turntable_Axis.Position[20].Vel := 0;
   PRODUCT_TYPE[2].Motion.Shaft_Scan_Turntable_Axis.Position[20].Pos := 0;
   PRODUCT_TYPE[2].Motion.Shaft_Scan_Turntable_Axis.Position[20].Vel := 0;
   PRODUCT_TYPE[3].Motion.Shaft_Scan_Turntable_Axis.Position[20].Pos := 0;
   PRODUCT_TYPE[3].Motion.Shaft_Scan_Turntable_Axis.Position[20].Vel := 0;
   PRODUCT_TYPE[4].Motion.Shaft_Scan_Turntable_Axis.Position[20].Pos := 0;
   PRODUCT_TYPE[4].Motion.Shaft_Scan_Turntable_Axis.Position[20].Vel := 0;
   PRODUCT_TYPE[5].Motion.Shaft_Scan_Turntable_Axis.Position[20].Pos := 0;
   PRODUCT_TYPE[5].Motion.Shaft_Scan_Turntable_Axis.Position[20].Vel := 0;
   PRODUCT_TYPE[6].Motion.Shaft_Scan_Turntable_Axis.Position[20].Pos := 0;
   PRODUCT_TYPE[6].Motion.Shaft_Scan_Turntable_Axis.Position[20].Vel := 0;
   PRODUCT_TYPE[7].Motion.Shaft_Scan_Turntable_Axis.Position[20].Pos := 0;
   PRODUCT_TYPE[7].Motion.Shaft_Scan_Turntable_Axis.Position[20].Vel := 0;
   PRODUCT_TYPE[8].Motion.Shaft_Scan_Turntable_Axis.Position[20].Pos := 0;
   PRODUCT_TYPE[8].Motion.Shaft_Scan_Turntable_Axis.Position[20].Vel := 0;
   PRODUCT_TYPE[9].Motion.Shaft_Scan_Turntable_Axis.Position[20].Pos := 0;
   PRODUCT_TYPE[9].Motion.Shaft_Scan_Turntable_Axis.Position[20].Vel := 0;
   PRODUCT_TYPE[10].Motion.Shaft_Scan_Turntable_Axis.Position[20].Pos := 0;
   PRODUCT_TYPE[10].Motion.Shaft_Scan_Turntable_Axis.Position[20].Vel := 0;
   PRODUCT_TYPE[1].Motion.Gluing_Rotary_Jig_Axis.Position[1].Pos := 0;
   PRODUCT_TYPE[1].Motion.Gluing_Rotary_Jig_Axis.Position[1].Vel := 20000;
   PRODUCT_TYPE[2].Motion.Gluing_Rotary_Jig_Axis.Position[1].Pos := 0;
   PRODUCT_TYPE[2].Motion.Gluing_Rotary_Jig_Axis.Position[1].Vel := 20000;
   PRODUCT_TYPE[3].Motion.Gluing_Rotary_Jig_Axis.Position[1].Pos := 0;
   PRODUCT_TYPE[3].Motion.Gluing_Rotary_Jig_Axis.Position[1].Vel := 20000;
   PRODUCT_TYPE[4].Motion.Gluing_Rotary_Jig_Axis.Position[1].Pos := 0;
   PRODUCT_TYPE[4].Motion.Gluing_Rotary_Jig_Axis.Position[1].Vel := 20000;
   PRODUCT_TYPE[5].Motion.Gluing_Rotary_Jig_Axis.Position[1].Pos := 0;
   PRODUCT_TYPE[5].Motion.Gluing_Rotary_Jig_Axis.Position[1].Vel := 20000;
   PRODUCT_TYPE[6].Motion.Gluing_Rotary_Jig_Axis.Position[1].Pos := 0;
   PRODUCT_TYPE[6].Motion.Gluing_Rotary_Jig_Axis.Position[1].Vel := 20000;
   PRODUCT_TYPE[7].Motion.Gluing_Rotary_Jig_Axis.Position[1].Pos := 0;
   PRODUCT_TYPE[7].Motion.Gluing_Rotary_Jig_Axis.Position[1].Vel := 20000;
   PRODUCT_TYPE[8].Motion.Gluing_Rotary_Jig_Axis.Position[1].Pos := 0;
   PRODUCT_TYPE[8].Motion.Gluing_Rotary_Jig_Axis.Position[1].Vel := 20000;
   PRODUCT_TYPE[9].Motion.Gluing_Rotary_Jig_Axis.Position[1].Pos := 0;
   PRODUCT_TYPE[9].Motion.Gluing_Rotary_Jig_Axis.Position[1].Vel := 20000;
   PRODUCT_TYPE[10].Motion.Gluing_Rotary_Jig_Axis.Position[1].Pos := 0;
   PRODUCT_TYPE[10].Motion.Gluing_Rotary_Jig_Axis.Position[1].Vel := 20000;
   PRODUCT_TYPE[1].Motion.Gluing_Rotary_Jig_Axis.Position[2].Pos := 0;
   PRODUCT_TYPE[1].Motion.Gluing_Rotary_Jig_Axis.Position[2].Vel := 20000;
   PRODUCT_TYPE[2].Motion.Gluing_Rotary_Jig_Axis.Position[2].Pos := 0;
   PRODUCT_TYPE[2].Motion.Gluing_Rotary_Jig_Axis.Position[2].Vel := 20000;
   PRODUCT_TYPE[3].Motion.Gluing_Rotary_Jig_Axis.Position[2].Pos := 0;
   PRODUCT_TYPE[3].Motion.Gluing_Rotary_Jig_Axis.Position[2].Vel := 20000;
   PRODUCT_TYPE[4].Motion.Gluing_Rotary_Jig_Axis.Position[2].Pos := 0;
   PRODUCT_TYPE[4].Motion.Gluing_Rotary_Jig_Axis.Position[2].Vel := 20000;
   PRODUCT_TYPE[5].Motion.Gluing_Rotary_Jig_Axis.Position[2].Pos := 0;
   PRODUCT_TYPE[5].Motion.Gluing_Rotary_Jig_Axis.Position[2].Vel := 20000;
   PRODUCT_TYPE[6].Motion.Gluing_Rotary_Jig_Axis.Position[2].Pos := 0;
   PRODUCT_TYPE[6].Motion.Gluing_Rotary_Jig_Axis.Position[2].Vel := 20000;
   PRODUCT_TYPE[7].Motion.Gluing_Rotary_Jig_Axis.Position[2].Pos := 0;
   PRODUCT_TYPE[7].Motion.Gluing_Rotary_Jig_Axis.Position[2].Vel := 20000;
   PRODUCT_TYPE[8].Motion.Gluing_Rotary_Jig_Axis.Position[2].Pos := 0;
   PRODUCT_TYPE[8].Motion.Gluing_Rotary_Jig_Axis.Position[2].Vel := 20000;
   PRODUCT_TYPE[9].Motion.Gluing_Rotary_Jig_Axis.Position[2].Pos := 0;
   PRODUCT_TYPE[9].Motion.Gluing_Rotary_Jig_Axis.Position[2].Vel := 20000;
   PRODUCT_TYPE[10].Motion.Gluing_Rotary_Jig_Axis.Position[2].Pos := 0;
   PRODUCT_TYPE[10].Motion.Gluing_Rotary_Jig_Axis.Position[2].Vel := 20000;
   PRODUCT_TYPE[1].Motion.Gluing_Rotary_Jig_Axis.Position[3].Pos := 680000;
   PRODUCT_TYPE[1].Motion.Gluing_Rotary_Jig_Axis.Position[3].Vel := 10000;
   PRODUCT_TYPE[2].Motion.Gluing_Rotary_Jig_Axis.Position[3].Pos := 680000;
   PRODUCT_TYPE[2].Motion.Gluing_Rotary_Jig_Axis.Position[3].Vel := 10000;
   PRODUCT_TYPE[3].Motion.Gluing_Rotary_Jig_Axis.Position[3].Pos := 680000;
   PRODUCT_TYPE[3].Motion.Gluing_Rotary_Jig_Axis.Position[3].Vel := 10000;
   PRODUCT_TYPE[4].Motion.Gluing_Rotary_Jig_Axis.Position[3].Pos := 680000;
   PRODUCT_TYPE[4].Motion.Gluing_Rotary_Jig_Axis.Position[3].Vel := 10000;
   PRODUCT_TYPE[5].Motion.Gluing_Rotary_Jig_Axis.Position[3].Pos := 680000;
   PRODUCT_TYPE[5].Motion.Gluing_Rotary_Jig_Axis.Position[3].Vel := 10000;
   PRODUCT_TYPE[6].Motion.Gluing_Rotary_Jig_Axis.Position[3].Pos := 680000;
   PRODUCT_TYPE[6].Motion.Gluing_Rotary_Jig_Axis.Position[3].Vel := 10000;
   PRODUCT_TYPE[7].Motion.Gluing_Rotary_Jig_Axis.Position[3].Pos := 680000;
   PRODUCT_TYPE[7].Motion.Gluing_Rotary_Jig_Axis.Position[3].Vel := 10000;
   PRODUCT_TYPE[8].Motion.Gluing_Rotary_Jig_Axis.Position[3].Pos := 680000;
   PRODUCT_TYPE[8].Motion.Gluing_Rotary_Jig_Axis.Position[3].Vel := 10000;
   PRODUCT_TYPE[9].Motion.Gluing_Rotary_Jig_Axis.Position[3].Pos := 680000;
   PRODUCT_TYPE[9].Motion.Gluing_Rotary_Jig_Axis.Position[3].Vel := 10000;
   PRODUCT_TYPE[10].Motion.Gluing_Rotary_Jig_Axis.Position[3].Pos := 680000;
   PRODUCT_TYPE[10].Motion.Gluing_Rotary_Jig_Axis.Position[3].Vel := 10000;
   PRODUCT_TYPE[1].Motion.Gluing_Rotary_Jig_Axis.Position[4].Pos := 680000;
   PRODUCT_TYPE[1].Motion.Gluing_Rotary_Jig_Axis.Position[4].Vel := 10000;
   PRODUCT_TYPE[2].Motion.Gluing_Rotary_Jig_Axis.Position[4].Pos := 680000;
   PRODUCT_TYPE[2].Motion.Gluing_Rotary_Jig_Axis.Position[4].Vel := 10000;
   PRODUCT_TYPE[3].Motion.Gluing_Rotary_Jig_Axis.Position[4].Pos := 680000;
   PRODUCT_TYPE[3].Motion.Gluing_Rotary_Jig_Axis.Position[4].Vel := 10000;
   PRODUCT_TYPE[4].Motion.Gluing_Rotary_Jig_Axis.Position[4].Pos := 680000;
   PRODUCT_TYPE[4].Motion.Gluing_Rotary_Jig_Axis.Position[4].Vel := 10000;
   PRODUCT_TYPE[5].Motion.Gluing_Rotary_Jig_Axis.Position[4].Pos := 680000;
   PRODUCT_TYPE[5].Motion.Gluing_Rotary_Jig_Axis.Position[4].Vel := 10000;
   PRODUCT_TYPE[6].Motion.Gluing_Rotary_Jig_Axis.Position[4].Pos := 680000;
   PRODUCT_TYPE[6].Motion.Gluing_Rotary_Jig_Axis.Position[4].Vel := 10000;
   PRODUCT_TYPE[7].Motion.Gluing_Rotary_Jig_Axis.Position[4].Pos := 680000;
   PRODUCT_TYPE[7].Motion.Gluing_Rotary_Jig_Axis.Position[4].Vel := 10000;
   PRODUCT_TYPE[8].Motion.Gluing_Rotary_Jig_Axis.Position[4].Pos := 680000;
   PRODUCT_TYPE[8].Motion.Gluing_Rotary_Jig_Axis.Position[4].Vel := 10000;
   PRODUCT_TYPE[9].Motion.Gluing_Rotary_Jig_Axis.Position[4].Pos := 680000;
   PRODUCT_TYPE[9].Motion.Gluing_Rotary_Jig_Axis.Position[4].Vel := 10000;
   PRODUCT_TYPE[10].Motion.Gluing_Rotary_Jig_Axis.Position[4].Pos := 680000;
   PRODUCT_TYPE[10].Motion.Gluing_Rotary_Jig_Axis.Position[4].Vel := 10000;
   PRODUCT_TYPE[1].Motion.Gluing_Rotary_Jig_Axis.Position[5].Pos := 680000;
   PRODUCT_TYPE[1].Motion.Gluing_Rotary_Jig_Axis.Position[5].Vel := 10000;
   PRODUCT_TYPE[2].Motion.Gluing_Rotary_Jig_Axis.Position[5].Pos := 680000;
   PRODUCT_TYPE[2].Motion.Gluing_Rotary_Jig_Axis.Position[5].Vel := 10000;
   PRODUCT_TYPE[3].Motion.Gluing_Rotary_Jig_Axis.Position[5].Pos := 680000;
   PRODUCT_TYPE[3].Motion.Gluing_Rotary_Jig_Axis.Position[5].Vel := 10000;
   PRODUCT_TYPE[4].Motion.Gluing_Rotary_Jig_Axis.Position[5].Pos := 680000;
   PRODUCT_TYPE[4].Motion.Gluing_Rotary_Jig_Axis.Position[5].Vel := 10000;
   PRODUCT_TYPE[5].Motion.Gluing_Rotary_Jig_Axis.Position[5].Pos := 680000;
   PRODUCT_TYPE[5].Motion.Gluing_Rotary_Jig_Axis.Position[5].Vel := 10000;
   PRODUCT_TYPE[6].Motion.Gluing_Rotary_Jig_Axis.Position[5].Pos := 680000;
   PRODUCT_TYPE[6].Motion.Gluing_Rotary_Jig_Axis.Position[5].Vel := 10000;
   PRODUCT_TYPE[7].Motion.Gluing_Rotary_Jig_Axis.Position[5].Pos := 680000;
   PRODUCT_TYPE[7].Motion.Gluing_Rotary_Jig_Axis.Position[5].Vel := 10000;
   PRODUCT_TYPE[8].Motion.Gluing_Rotary_Jig_Axis.Position[5].Pos := 680000;
   PRODUCT_TYPE[8].Motion.Gluing_Rotary_Jig_Axis.Position[5].Vel := 10000;
   PRODUCT_TYPE[9].Motion.Gluing_Rotary_Jig_Axis.Position[5].Pos := 680000;
   PRODUCT_TYPE[9].Motion.Gluing_Rotary_Jig_Axis.Position[5].Vel := 10000;
   PRODUCT_TYPE[10].Motion.Gluing_Rotary_Jig_Axis.Position[5].Pos := 680000;
   PRODUCT_TYPE[10].Motion.Gluing_Rotary_Jig_Axis.Position[5].Vel := 10000;
   PRODUCT_TYPE[1].Motion.Gluing_Rotary_Jig_Axis.Position[6].Pos := 680000;
   PRODUCT_TYPE[1].Motion.Gluing_Rotary_Jig_Axis.Position[6].Vel := 10000;
   PRODUCT_TYPE[2].Motion.Gluing_Rotary_Jig_Axis.Position[6].Pos := 680000;
   PRODUCT_TYPE[2].Motion.Gluing_Rotary_Jig_Axis.Position[6].Vel := 10000;
   PRODUCT_TYPE[3].Motion.Gluing_Rotary_Jig_Axis.Position[6].Pos := 680000;
   PRODUCT_TYPE[3].Motion.Gluing_Rotary_Jig_Axis.Position[6].Vel := 10000;
   PRODUCT_TYPE[4].Motion.Gluing_Rotary_Jig_Axis.Position[6].Pos := 680000;
   PRODUCT_TYPE[4].Motion.Gluing_Rotary_Jig_Axis.Position[6].Vel := 10000;
   PRODUCT_TYPE[5].Motion.Gluing_Rotary_Jig_Axis.Position[6].Pos := 680000;
   PRODUCT_TYPE[5].Motion.Gluing_Rotary_Jig_Axis.Position[6].Vel := 10000;
   PRODUCT_TYPE[6].Motion.Gluing_Rotary_Jig_Axis.Position[6].Pos := 680000;
   PRODUCT_TYPE[6].Motion.Gluing_Rotary_Jig_Axis.Position[6].Vel := 10000;
   PRODUCT_TYPE[7].Motion.Gluing_Rotary_Jig_Axis.Position[6].Pos := 680000;
   PRODUCT_TYPE[7].Motion.Gluing_Rotary_Jig_Axis.Position[6].Vel := 10000;
   PRODUCT_TYPE[8].Motion.Gluing_Rotary_Jig_Axis.Position[6].Pos := 680000;
   PRODUCT_TYPE[8].Motion.Gluing_Rotary_Jig_Axis.Position[6].Vel := 10000;
   PRODUCT_TYPE[9].Motion.Gluing_Rotary_Jig_Axis.Position[6].Pos := 680000;
   PRODUCT_TYPE[9].Motion.Gluing_Rotary_Jig_Axis.Position[6].Vel := 10000;
   PRODUCT_TYPE[10].Motion.Gluing_Rotary_Jig_Axis.Position[6].Pos := 680000;
   PRODUCT_TYPE[10].Motion.Gluing_Rotary_Jig_Axis.Position[6].Vel := 10000;
   PRODUCT_TYPE[1].Motion.Gluing_Rotary_Jig_Axis.Position[7].Pos := 90000;
   PRODUCT_TYPE[1].Motion.Gluing_Rotary_Jig_Axis.Position[7].Vel := 10000;
   PRODUCT_TYPE[2].Motion.Gluing_Rotary_Jig_Axis.Position[7].Pos := 90000;
   PRODUCT_TYPE[2].Motion.Gluing_Rotary_Jig_Axis.Position[7].Vel := 10000;
   PRODUCT_TYPE[3].Motion.Gluing_Rotary_Jig_Axis.Position[7].Pos := 90000;
   PRODUCT_TYPE[3].Motion.Gluing_Rotary_Jig_Axis.Position[7].Vel := 10000;
   PRODUCT_TYPE[4].Motion.Gluing_Rotary_Jig_Axis.Position[7].Pos := 90000;
   PRODUCT_TYPE[4].Motion.Gluing_Rotary_Jig_Axis.Position[7].Vel := 10000;
   PRODUCT_TYPE[5].Motion.Gluing_Rotary_Jig_Axis.Position[7].Pos := 90000;
   PRODUCT_TYPE[5].Motion.Gluing_Rotary_Jig_Axis.Position[7].Vel := 10000;
   PRODUCT_TYPE[6].Motion.Gluing_Rotary_Jig_Axis.Position[7].Pos := 90000;
   PRODUCT_TYPE[6].Motion.Gluing_Rotary_Jig_Axis.Position[7].Vel := 10000;
   PRODUCT_TYPE[7].Motion.Gluing_Rotary_Jig_Axis.Position[7].Pos := 90000;
   PRODUCT_TYPE[7].Motion.Gluing_Rotary_Jig_Axis.Position[7].Vel := 10000;
   PRODUCT_TYPE[8].Motion.Gluing_Rotary_Jig_Axis.Position[7].Pos := 90000;
   PRODUCT_TYPE[8].Motion.Gluing_Rotary_Jig_Axis.Position[7].Vel := 10000;
   PRODUCT_TYPE[9].Motion.Gluing_Rotary_Jig_Axis.Position[7].Pos := 90000;
   PRODUCT_TYPE[9].Motion.Gluing_Rotary_Jig_Axis.Position[7].Vel := 10000;
   PRODUCT_TYPE[10].Motion.Gluing_Rotary_Jig_Axis.Position[7].Pos := 90000;
   PRODUCT_TYPE[10].Motion.Gluing_Rotary_Jig_Axis.Position[7].Vel := 10000;
   PRODUCT_TYPE[1].Motion.Gluing_Rotary_Jig_Axis.Position[8].Pos := 180000;
   PRODUCT_TYPE[1].Motion.Gluing_Rotary_Jig_Axis.Position[8].Vel := 10000;
   PRODUCT_TYPE[2].Motion.Gluing_Rotary_Jig_Axis.Position[8].Pos := 180000;
   PRODUCT_TYPE[2].Motion.Gluing_Rotary_Jig_Axis.Position[8].Vel := 10000;
   PRODUCT_TYPE[3].Motion.Gluing_Rotary_Jig_Axis.Position[8].Pos := 180000;
   PRODUCT_TYPE[3].Motion.Gluing_Rotary_Jig_Axis.Position[8].Vel := 10000;
   PRODUCT_TYPE[4].Motion.Gluing_Rotary_Jig_Axis.Position[8].Pos := 180000;
   PRODUCT_TYPE[4].Motion.Gluing_Rotary_Jig_Axis.Position[8].Vel := 10000;
   PRODUCT_TYPE[5].Motion.Gluing_Rotary_Jig_Axis.Position[8].Pos := 180000;
   PRODUCT_TYPE[5].Motion.Gluing_Rotary_Jig_Axis.Position[8].Vel := 10000;
   PRODUCT_TYPE[6].Motion.Gluing_Rotary_Jig_Axis.Position[8].Pos := 180000;
   PRODUCT_TYPE[6].Motion.Gluing_Rotary_Jig_Axis.Position[8].Vel := 10000;
   PRODUCT_TYPE[7].Motion.Gluing_Rotary_Jig_Axis.Position[8].Pos := 180000;
   PRODUCT_TYPE[7].Motion.Gluing_Rotary_Jig_Axis.Position[8].Vel := 10000;
   PRODUCT_TYPE[8].Motion.Gluing_Rotary_Jig_Axis.Position[8].Pos := 180000;
   PRODUCT_TYPE[8].Motion.Gluing_Rotary_Jig_Axis.Position[8].Vel := 10000;
   PRODUCT_TYPE[9].Motion.Gluing_Rotary_Jig_Axis.Position[8].Pos := 180000;
   PRODUCT_TYPE[9].Motion.Gluing_Rotary_Jig_Axis.Position[8].Vel := 10000;
   PRODUCT_TYPE[10].Motion.Gluing_Rotary_Jig_Axis.Position[8].Pos := 180000;
   PRODUCT_TYPE[10].Motion.Gluing_Rotary_Jig_Axis.Position[8].Vel := 10000;
   PRODUCT_TYPE[1].Motion.Gluing_Rotary_Jig_Axis.Position[9].Pos := 270000;
   PRODUCT_TYPE[1].Motion.Gluing_Rotary_Jig_Axis.Position[9].Vel := 10000;
   PRODUCT_TYPE[2].Motion.Gluing_Rotary_Jig_Axis.Position[9].Pos := 270000;
   PRODUCT_TYPE[2].Motion.Gluing_Rotary_Jig_Axis.Position[9].Vel := 10000;
   PRODUCT_TYPE[3].Motion.Gluing_Rotary_Jig_Axis.Position[9].Pos := 270000;
   PRODUCT_TYPE[3].Motion.Gluing_Rotary_Jig_Axis.Position[9].Vel := 10000;
   PRODUCT_TYPE[4].Motion.Gluing_Rotary_Jig_Axis.Position[9].Pos := 270000;
   PRODUCT_TYPE[4].Motion.Gluing_Rotary_Jig_Axis.Position[9].Vel := 10000;
   PRODUCT_TYPE[5].Motion.Gluing_Rotary_Jig_Axis.Position[9].Pos := 270000;
   PRODUCT_TYPE[5].Motion.Gluing_Rotary_Jig_Axis.Position[9].Vel := 10000;
   PRODUCT_TYPE[6].Motion.Gluing_Rotary_Jig_Axis.Position[9].Pos := 270000;
   PRODUCT_TYPE[6].Motion.Gluing_Rotary_Jig_Axis.Position[9].Vel := 10000;
   PRODUCT_TYPE[7].Motion.Gluing_Rotary_Jig_Axis.Position[9].Pos := 270000;
   PRODUCT_TYPE[7].Motion.Gluing_Rotary_Jig_Axis.Position[9].Vel := 10000;
   PRODUCT_TYPE[8].Motion.Gluing_Rotary_Jig_Axis.Position[9].Pos := 270000;
   PRODUCT_TYPE[8].Motion.Gluing_Rotary_Jig_Axis.Position[9].Vel := 10000;
   PRODUCT_TYPE[9].Motion.Gluing_Rotary_Jig_Axis.Position[9].Pos := 270000;
   PRODUCT_TYPE[9].Motion.Gluing_Rotary_Jig_Axis.Position[9].Vel := 10000;
   PRODUCT_TYPE[10].Motion.Gluing_Rotary_Jig_Axis.Position[9].Pos := 270000;
   PRODUCT_TYPE[10].Motion.Gluing_Rotary_Jig_Axis.Position[9].Vel := 10000;
   PRODUCT_TYPE[1].Motion.Gluing_Rotary_Jig_Axis.Position[10].Pos := 0;
   PRODUCT_TYPE[1].Motion.Gluing_Rotary_Jig_Axis.Position[10].Vel := 0;
   PRODUCT_TYPE[2].Motion.Gluing_Rotary_Jig_Axis.Position[10].Pos := 0;
   PRODUCT_TYPE[2].Motion.Gluing_Rotary_Jig_Axis.Position[10].Vel := 0;
   PRODUCT_TYPE[3].Motion.Gluing_Rotary_Jig_Axis.Position[10].Pos := 0;
   PRODUCT_TYPE[3].Motion.Gluing_Rotary_Jig_Axis.Position[10].Vel := 0;
   PRODUCT_TYPE[4].Motion.Gluing_Rotary_Jig_Axis.Position[10].Pos := 0;
   PRODUCT_TYPE[4].Motion.Gluing_Rotary_Jig_Axis.Position[10].Vel := 0;
   PRODUCT_TYPE[5].Motion.Gluing_Rotary_Jig_Axis.Position[10].Pos := 0;
   PRODUCT_TYPE[5].Motion.Gluing_Rotary_Jig_Axis.Position[10].Vel := 0;
   PRODUCT_TYPE[6].Motion.Gluing_Rotary_Jig_Axis.Position[10].Pos := 0;
   PRODUCT_TYPE[6].Motion.Gluing_Rotary_Jig_Axis.Position[10].Vel := 0;
   PRODUCT_TYPE[7].Motion.Gluing_Rotary_Jig_Axis.Position[10].Pos := 0;
   PRODUCT_TYPE[7].Motion.Gluing_Rotary_Jig_Axis.Position[10].Vel := 0;
   PRODUCT_TYPE[8].Motion.Gluing_Rotary_Jig_Axis.Position[10].Pos := 0;
   PRODUCT_TYPE[8].Motion.Gluing_Rotary_Jig_Axis.Position[10].Vel := 0;
   PRODUCT_TYPE[9].Motion.Gluing_Rotary_Jig_Axis.Position[10].Pos := 0;
   PRODUCT_TYPE[9].Motion.Gluing_Rotary_Jig_Axis.Position[10].Vel := 0;
   PRODUCT_TYPE[10].Motion.Gluing_Rotary_Jig_Axis.Position[10].Pos := 0;
   PRODUCT_TYPE[10].Motion.Gluing_Rotary_Jig_Axis.Position[10].Vel := 0;
   PRODUCT_TYPE[1].Motion.Gluing_Rotary_Jig_Axis.Position[11].Pos := 0;
   PRODUCT_TYPE[1].Motion.Gluing_Rotary_Jig_Axis.Position[11].Vel := 0;
   PRODUCT_TYPE[2].Motion.Gluing_Rotary_Jig_Axis.Position[11].Pos := 0;
   PRODUCT_TYPE[2].Motion.Gluing_Rotary_Jig_Axis.Position[11].Vel := 0;
   PRODUCT_TYPE[3].Motion.Gluing_Rotary_Jig_Axis.Position[11].Pos := 0;
   PRODUCT_TYPE[3].Motion.Gluing_Rotary_Jig_Axis.Position[11].Vel := 0;
   PRODUCT_TYPE[4].Motion.Gluing_Rotary_Jig_Axis.Position[11].Pos := 0;
   PRODUCT_TYPE[4].Motion.Gluing_Rotary_Jig_Axis.Position[11].Vel := 0;
   PRODUCT_TYPE[5].Motion.Gluing_Rotary_Jig_Axis.Position[11].Pos := 0;
   PRODUCT_TYPE[5].Motion.Gluing_Rotary_Jig_Axis.Position[11].Vel := 0;
   PRODUCT_TYPE[6].Motion.Gluing_Rotary_Jig_Axis.Position[11].Pos := 0;
   PRODUCT_TYPE[6].Motion.Gluing_Rotary_Jig_Axis.Position[11].Vel := 0;
   PRODUCT_TYPE[7].Motion.Gluing_Rotary_Jig_Axis.Position[11].Pos := 0;
   PRODUCT_TYPE[7].Motion.Gluing_Rotary_Jig_Axis.Position[11].Vel := 0;
   PRODUCT_TYPE[8].Motion.Gluing_Rotary_Jig_Axis.Position[11].Pos := 0;
   PRODUCT_TYPE[8].Motion.Gluing_Rotary_Jig_Axis.Position[11].Vel := 0;
   PRODUCT_TYPE[9].Motion.Gluing_Rotary_Jig_Axis.Position[11].Pos := 0;
   PRODUCT_TYPE[9].Motion.Gluing_Rotary_Jig_Axis.Position[11].Vel := 0;
   PRODUCT_TYPE[10].Motion.Gluing_Rotary_Jig_Axis.Position[11].Pos := 0;
   PRODUCT_TYPE[10].Motion.Gluing_Rotary_Jig_Axis.Position[11].Vel := 0;
   PRODUCT_TYPE[1].Motion.Gluing_Rotary_Jig_Axis.Position[12].Pos := 0;
   PRODUCT_TYPE[1].Motion.Gluing_Rotary_Jig_Axis.Position[12].Vel := 0;
   PRODUCT_TYPE[2].Motion.Gluing_Rotary_Jig_Axis.Position[12].Pos := 0;
   PRODUCT_TYPE[2].Motion.Gluing_Rotary_Jig_Axis.Position[12].Vel := 0;
   PRODUCT_TYPE[3].Motion.Gluing_Rotary_Jig_Axis.Position[12].Pos := 0;
   PRODUCT_TYPE[3].Motion.Gluing_Rotary_Jig_Axis.Position[12].Vel := 0;
   PRODUCT_TYPE[4].Motion.Gluing_Rotary_Jig_Axis.Position[12].Pos := 0;
   PRODUCT_TYPE[4].Motion.Gluing_Rotary_Jig_Axis.Position[12].Vel := 0;
   PRODUCT_TYPE[5].Motion.Gluing_Rotary_Jig_Axis.Position[12].Pos := 0;
   PRODUCT_TYPE[5].Motion.Gluing_Rotary_Jig_Axis.Position[12].Vel := 0;
   PRODUCT_TYPE[6].Motion.Gluing_Rotary_Jig_Axis.Position[12].Pos := 0;
   PRODUCT_TYPE[6].Motion.Gluing_Rotary_Jig_Axis.Position[12].Vel := 0;
   PRODUCT_TYPE[7].Motion.Gluing_Rotary_Jig_Axis.Position[12].Pos := 0;
   PRODUCT_TYPE[7].Motion.Gluing_Rotary_Jig_Axis.Position[12].Vel := 0;
   PRODUCT_TYPE[8].Motion.Gluing_Rotary_Jig_Axis.Position[12].Pos := 0;
   PRODUCT_TYPE[8].Motion.Gluing_Rotary_Jig_Axis.Position[12].Vel := 0;
   PRODUCT_TYPE[9].Motion.Gluing_Rotary_Jig_Axis.Position[12].Pos := 0;
   PRODUCT_TYPE[9].Motion.Gluing_Rotary_Jig_Axis.Position[12].Vel := 0;
   PRODUCT_TYPE[10].Motion.Gluing_Rotary_Jig_Axis.Position[12].Pos := 0;
   PRODUCT_TYPE[10].Motion.Gluing_Rotary_Jig_Axis.Position[12].Vel := 0;
   PRODUCT_TYPE[1].Motion.Gluing_Rotary_Jig_Axis.Position[13].Pos := 0;
   PRODUCT_TYPE[1].Motion.Gluing_Rotary_Jig_Axis.Position[13].Vel := 0;
   PRODUCT_TYPE[2].Motion.Gluing_Rotary_Jig_Axis.Position[13].Pos := 0;
   PRODUCT_TYPE[2].Motion.Gluing_Rotary_Jig_Axis.Position[13].Vel := 0;
   PRODUCT_TYPE[3].Motion.Gluing_Rotary_Jig_Axis.Position[13].Pos := 0;
   PRODUCT_TYPE[3].Motion.Gluing_Rotary_Jig_Axis.Position[13].Vel := 0;
   PRODUCT_TYPE[4].Motion.Gluing_Rotary_Jig_Axis.Position[13].Pos := 0;
   PRODUCT_TYPE[4].Motion.Gluing_Rotary_Jig_Axis.Position[13].Vel := 0;
   PRODUCT_TYPE[5].Motion.Gluing_Rotary_Jig_Axis.Position[13].Pos := 0;
   PRODUCT_TYPE[5].Motion.Gluing_Rotary_Jig_Axis.Position[13].Vel := 0;
   PRODUCT_TYPE[6].Motion.Gluing_Rotary_Jig_Axis.Position[13].Pos := 0;
   PRODUCT_TYPE[6].Motion.Gluing_Rotary_Jig_Axis.Position[13].Vel := 0;
   PRODUCT_TYPE[7].Motion.Gluing_Rotary_Jig_Axis.Position[13].Pos := 0;
   PRODUCT_TYPE[7].Motion.Gluing_Rotary_Jig_Axis.Position[13].Vel := 0;
   PRODUCT_TYPE[8].Motion.Gluing_Rotary_Jig_Axis.Position[13].Pos := 0;
   PRODUCT_TYPE[8].Motion.Gluing_Rotary_Jig_Axis.Position[13].Vel := 0;
   PRODUCT_TYPE[9].Motion.Gluing_Rotary_Jig_Axis.Position[13].Pos := 0;
   PRODUCT_TYPE[9].Motion.Gluing_Rotary_Jig_Axis.Position[13].Vel := 0;
   PRODUCT_TYPE[10].Motion.Gluing_Rotary_Jig_Axis.Position[13].Pos := 0;
   PRODUCT_TYPE[10].Motion.Gluing_Rotary_Jig_Axis.Position[13].Vel := 0;
   PRODUCT_TYPE[1].Motion.Gluing_Rotary_Jig_Axis.Position[14].Pos := 0;
   PRODUCT_TYPE[1].Motion.Gluing_Rotary_Jig_Axis.Position[14].Vel := 0;
   PRODUCT_TYPE[2].Motion.Gluing_Rotary_Jig_Axis.Position[14].Pos := 0;
   PRODUCT_TYPE[2].Motion.Gluing_Rotary_Jig_Axis.Position[14].Vel := 0;
   PRODUCT_TYPE[3].Motion.Gluing_Rotary_Jig_Axis.Position[14].Pos := 0;
   PRODUCT_TYPE[3].Motion.Gluing_Rotary_Jig_Axis.Position[14].Vel := 0;
   PRODUCT_TYPE[4].Motion.Gluing_Rotary_Jig_Axis.Position[14].Pos := 0;
   PRODUCT_TYPE[4].Motion.Gluing_Rotary_Jig_Axis.Position[14].Vel := 0;
   PRODUCT_TYPE[5].Motion.Gluing_Rotary_Jig_Axis.Position[14].Pos := 0;
   PRODUCT_TYPE[5].Motion.Gluing_Rotary_Jig_Axis.Position[14].Vel := 0;
   PRODUCT_TYPE[6].Motion.Gluing_Rotary_Jig_Axis.Position[14].Pos := 0;
   PRODUCT_TYPE[6].Motion.Gluing_Rotary_Jig_Axis.Position[14].Vel := 0;
   PRODUCT_TYPE[7].Motion.Gluing_Rotary_Jig_Axis.Position[14].Pos := 0;
   PRODUCT_TYPE[7].Motion.Gluing_Rotary_Jig_Axis.Position[14].Vel := 0;
   PRODUCT_TYPE[8].Motion.Gluing_Rotary_Jig_Axis.Position[14].Pos := 0;
   PRODUCT_TYPE[8].Motion.Gluing_Rotary_Jig_Axis.Position[14].Vel := 0;
   PRODUCT_TYPE[9].Motion.Gluing_Rotary_Jig_Axis.Position[14].Pos := 0;
   PRODUCT_TYPE[9].Motion.Gluing_Rotary_Jig_Axis.Position[14].Vel := 0;
   PRODUCT_TYPE[10].Motion.Gluing_Rotary_Jig_Axis.Position[14].Pos := 0;
   PRODUCT_TYPE[10].Motion.Gluing_Rotary_Jig_Axis.Position[14].Vel := 0;
   PRODUCT_TYPE[1].Motion.Gluing_Rotary_Jig_Axis.Position[15].Pos := 0;
   PRODUCT_TYPE[1].Motion.Gluing_Rotary_Jig_Axis.Position[15].Vel := 0;
   PRODUCT_TYPE[2].Motion.Gluing_Rotary_Jig_Axis.Position[15].Pos := 0;
   PRODUCT_TYPE[2].Motion.Gluing_Rotary_Jig_Axis.Position[15].Vel := 0;
   PRODUCT_TYPE[3].Motion.Gluing_Rotary_Jig_Axis.Position[15].Pos := 0;
   PRODUCT_TYPE[3].Motion.Gluing_Rotary_Jig_Axis.Position[15].Vel := 0;
   PRODUCT_TYPE[4].Motion.Gluing_Rotary_Jig_Axis.Position[15].Pos := 0;
   PRODUCT_TYPE[4].Motion.Gluing_Rotary_Jig_Axis.Position[15].Vel := 0;
   PRODUCT_TYPE[5].Motion.Gluing_Rotary_Jig_Axis.Position[15].Pos := 0;
   PRODUCT_TYPE[5].Motion.Gluing_Rotary_Jig_Axis.Position[15].Vel := 0;
   PRODUCT_TYPE[6].Motion.Gluing_Rotary_Jig_Axis.Position[15].Pos := 0;
   PRODUCT_TYPE[6].Motion.Gluing_Rotary_Jig_Axis.Position[15].Vel := 0;
   PRODUCT_TYPE[7].Motion.Gluing_Rotary_Jig_Axis.Position[15].Pos := 0;
   PRODUCT_TYPE[7].Motion.Gluing_Rotary_Jig_Axis.Position[15].Vel := 0;
   PRODUCT_TYPE[8].Motion.Gluing_Rotary_Jig_Axis.Position[15].Pos := 0;
   PRODUCT_TYPE[8].Motion.Gluing_Rotary_Jig_Axis.Position[15].Vel := 0;
   PRODUCT_TYPE[9].Motion.Gluing_Rotary_Jig_Axis.Position[15].Pos := 0;
   PRODUCT_TYPE[9].Motion.Gluing_Rotary_Jig_Axis.Position[15].Vel := 0;
   PRODUCT_TYPE[10].Motion.Gluing_Rotary_Jig_Axis.Position[15].Pos := 0;
   PRODUCT_TYPE[10].Motion.Gluing_Rotary_Jig_Axis.Position[15].Vel := 0;
   PRODUCT_TYPE[1].Motion.Gluing_Rotary_Jig_Axis.Position[16].Pos := 0;
   PRODUCT_TYPE[1].Motion.Gluing_Rotary_Jig_Axis.Position[16].Vel := 0;
   PRODUCT_TYPE[2].Motion.Gluing_Rotary_Jig_Axis.Position[16].Pos := 0;
   PRODUCT_TYPE[2].Motion.Gluing_Rotary_Jig_Axis.Position[16].Vel := 0;
   PRODUCT_TYPE[3].Motion.Gluing_Rotary_Jig_Axis.Position[16].Pos := 0;
   PRODUCT_TYPE[3].Motion.Gluing_Rotary_Jig_Axis.Position[16].Vel := 0;
   PRODUCT_TYPE[4].Motion.Gluing_Rotary_Jig_Axis.Position[16].Pos := 0;
   PRODUCT_TYPE[4].Motion.Gluing_Rotary_Jig_Axis.Position[16].Vel := 0;
   PRODUCT_TYPE[5].Motion.Gluing_Rotary_Jig_Axis.Position[16].Pos := 0;
   PRODUCT_TYPE[5].Motion.Gluing_Rotary_Jig_Axis.Position[16].Vel := 0;
   PRODUCT_TYPE[6].Motion.Gluing_Rotary_Jig_Axis.Position[16].Pos := 0;
   PRODUCT_TYPE[6].Motion.Gluing_Rotary_Jig_Axis.Position[16].Vel := 0;
   PRODUCT_TYPE[7].Motion.Gluing_Rotary_Jig_Axis.Position[16].Pos := 0;
   PRODUCT_TYPE[7].Motion.Gluing_Rotary_Jig_Axis.Position[16].Vel := 0;
   PRODUCT_TYPE[8].Motion.Gluing_Rotary_Jig_Axis.Position[16].Pos := 0;
   PRODUCT_TYPE[8].Motion.Gluing_Rotary_Jig_Axis.Position[16].Vel := 0;
   PRODUCT_TYPE[9].Motion.Gluing_Rotary_Jig_Axis.Position[16].Pos := 0;
   PRODUCT_TYPE[9].Motion.Gluing_Rotary_Jig_Axis.Position[16].Vel := 0;
   PRODUCT_TYPE[10].Motion.Gluing_Rotary_Jig_Axis.Position[16].Pos := 0;
   PRODUCT_TYPE[10].Motion.Gluing_Rotary_Jig_Axis.Position[16].Vel := 0;
   PRODUCT_TYPE[1].Motion.Gluing_Rotary_Jig_Axis.Position[17].Pos := 0;
   PRODUCT_TYPE[1].Motion.Gluing_Rotary_Jig_Axis.Position[17].Vel := 0;
   PRODUCT_TYPE[2].Motion.Gluing_Rotary_Jig_Axis.Position[17].Pos := 0;
   PRODUCT_TYPE[2].Motion.Gluing_Rotary_Jig_Axis.Position[17].Vel := 0;
   PRODUCT_TYPE[3].Motion.Gluing_Rotary_Jig_Axis.Position[17].Pos := 0;
   PRODUCT_TYPE[3].Motion.Gluing_Rotary_Jig_Axis.Position[17].Vel := 0;
   PRODUCT_TYPE[4].Motion.Gluing_Rotary_Jig_Axis.Position[17].Pos := 0;
   PRODUCT_TYPE[4].Motion.Gluing_Rotary_Jig_Axis.Position[17].Vel := 0;
   PRODUCT_TYPE[5].Motion.Gluing_Rotary_Jig_Axis.Position[17].Pos := 0;
   PRODUCT_TYPE[5].Motion.Gluing_Rotary_Jig_Axis.Position[17].Vel := 0;
   PRODUCT_TYPE[6].Motion.Gluing_Rotary_Jig_Axis.Position[17].Pos := 0;
   PRODUCT_TYPE[6].Motion.Gluing_Rotary_Jig_Axis.Position[17].Vel := 0;
   PRODUCT_TYPE[7].Motion.Gluing_Rotary_Jig_Axis.Position[17].Pos := 0;
   PRODUCT_TYPE[7].Motion.Gluing_Rotary_Jig_Axis.Position[17].Vel := 0;
   PRODUCT_TYPE[8].Motion.Gluing_Rotary_Jig_Axis.Position[17].Pos := 0;
   PRODUCT_TYPE[8].Motion.Gluing_Rotary_Jig_Axis.Position[17].Vel := 0;
   PRODUCT_TYPE[9].Motion.Gluing_Rotary_Jig_Axis.Position[17].Pos := 0;
   PRODUCT_TYPE[9].Motion.Gluing_Rotary_Jig_Axis.Position[17].Vel := 0;
   PRODUCT_TYPE[10].Motion.Gluing_Rotary_Jig_Axis.Position[17].Pos := 0;
   PRODUCT_TYPE[10].Motion.Gluing_Rotary_Jig_Axis.Position[17].Vel := 0;
   PRODUCT_TYPE[1].Motion.Gluing_Rotary_Jig_Axis.Position[18].Pos := 0;
   PRODUCT_TYPE[1].Motion.Gluing_Rotary_Jig_Axis.Position[18].Vel := 0;
   PRODUCT_TYPE[2].Motion.Gluing_Rotary_Jig_Axis.Position[18].Pos := 0;
   PRODUCT_TYPE[2].Motion.Gluing_Rotary_Jig_Axis.Position[18].Vel := 0;
   PRODUCT_TYPE[3].Motion.Gluing_Rotary_Jig_Axis.Position[18].Pos := 0;
   PRODUCT_TYPE[3].Motion.Gluing_Rotary_Jig_Axis.Position[18].Vel := 0;
   PRODUCT_TYPE[4].Motion.Gluing_Rotary_Jig_Axis.Position[18].Pos := 0;
   PRODUCT_TYPE[4].Motion.Gluing_Rotary_Jig_Axis.Position[18].Vel := 0;
   PRODUCT_TYPE[5].Motion.Gluing_Rotary_Jig_Axis.Position[18].Pos := 0;
   PRODUCT_TYPE[5].Motion.Gluing_Rotary_Jig_Axis.Position[18].Vel := 0;
   PRODUCT_TYPE[6].Motion.Gluing_Rotary_Jig_Axis.Position[18].Pos := 0;
   PRODUCT_TYPE[6].Motion.Gluing_Rotary_Jig_Axis.Position[18].Vel := 0;
   PRODUCT_TYPE[7].Motion.Gluing_Rotary_Jig_Axis.Position[18].Pos := 0;
   PRODUCT_TYPE[7].Motion.Gluing_Rotary_Jig_Axis.Position[18].Vel := 0;
   PRODUCT_TYPE[8].Motion.Gluing_Rotary_Jig_Axis.Position[18].Pos := 0;
   PRODUCT_TYPE[8].Motion.Gluing_Rotary_Jig_Axis.Position[18].Vel := 0;
   PRODUCT_TYPE[9].Motion.Gluing_Rotary_Jig_Axis.Position[18].Pos := 0;
   PRODUCT_TYPE[9].Motion.Gluing_Rotary_Jig_Axis.Position[18].Vel := 0;
   PRODUCT_TYPE[10].Motion.Gluing_Rotary_Jig_Axis.Position[18].Pos := 0;
   PRODUCT_TYPE[10].Motion.Gluing_Rotary_Jig_Axis.Position[18].Vel := 0;
   PRODUCT_TYPE[1].Motion.Gluing_Rotary_Jig_Axis.Position[19].Pos := 0;
   PRODUCT_TYPE[1].Motion.Gluing_Rotary_Jig_Axis.Position[19].Vel := 0;
   PRODUCT_TYPE[2].Motion.Gluing_Rotary_Jig_Axis.Position[19].Pos := 0;
   PRODUCT_TYPE[2].Motion.Gluing_Rotary_Jig_Axis.Position[19].Vel := 0;
   PRODUCT_TYPE[3].Motion.Gluing_Rotary_Jig_Axis.Position[19].Pos := 0;
   PRODUCT_TYPE[3].Motion.Gluing_Rotary_Jig_Axis.Position[19].Vel := 0;
   PRODUCT_TYPE[4].Motion.Gluing_Rotary_Jig_Axis.Position[19].Pos := 0;
   PRODUCT_TYPE[4].Motion.Gluing_Rotary_Jig_Axis.Position[19].Vel := 0;
   PRODUCT_TYPE[5].Motion.Gluing_Rotary_Jig_Axis.Position[19].Pos := 0;
   PRODUCT_TYPE[5].Motion.Gluing_Rotary_Jig_Axis.Position[19].Vel := 0;
   PRODUCT_TYPE[6].Motion.Gluing_Rotary_Jig_Axis.Position[19].Pos := 0;
   PRODUCT_TYPE[6].Motion.Gluing_Rotary_Jig_Axis.Position[19].Vel := 0;
   PRODUCT_TYPE[7].Motion.Gluing_Rotary_Jig_Axis.Position[19].Pos := 0;
   PRODUCT_TYPE[7].Motion.Gluing_Rotary_Jig_Axis.Position[19].Vel := 0;
   PRODUCT_TYPE[8].Motion.Gluing_Rotary_Jig_Axis.Position[19].Pos := 0;
   PRODUCT_TYPE[8].Motion.Gluing_Rotary_Jig_Axis.Position[19].Vel := 0;
   PRODUCT_TYPE[9].Motion.Gluing_Rotary_Jig_Axis.Position[19].Pos := 0;
   PRODUCT_TYPE[9].Motion.Gluing_Rotary_Jig_Axis.Position[19].Vel := 0;
   PRODUCT_TYPE[10].Motion.Gluing_Rotary_Jig_Axis.Position[19].Pos := 0;
   PRODUCT_TYPE[10].Motion.Gluing_Rotary_Jig_Axis.Position[19].Vel := 0;
   PRODUCT_TYPE[1].Motion.Gluing_Rotary_Jig_Axis.Position[20].Pos := 0;
   PRODUCT_TYPE[1].Motion.Gluing_Rotary_Jig_Axis.Position[20].Vel := 0;
   PRODUCT_TYPE[2].Motion.Gluing_Rotary_Jig_Axis.Position[20].Pos := 0;
   PRODUCT_TYPE[2].Motion.Gluing_Rotary_Jig_Axis.Position[20].Vel := 0;
   PRODUCT_TYPE[3].Motion.Gluing_Rotary_Jig_Axis.Position[20].Pos := 0;
   PRODUCT_TYPE[3].Motion.Gluing_Rotary_Jig_Axis.Position[20].Vel := 0;
   PRODUCT_TYPE[4].Motion.Gluing_Rotary_Jig_Axis.Position[20].Pos := 0;
   PRODUCT_TYPE[4].Motion.Gluing_Rotary_Jig_Axis.Position[20].Vel := 0;
   PRODUCT_TYPE[5].Motion.Gluing_Rotary_Jig_Axis.Position[20].Pos := 0;
   PRODUCT_TYPE[5].Motion.Gluing_Rotary_Jig_Axis.Position[20].Vel := 0;
   PRODUCT_TYPE[6].Motion.Gluing_Rotary_Jig_Axis.Position[20].Pos := 0;
   PRODUCT_TYPE[6].Motion.Gluing_Rotary_Jig_Axis.Position[20].Vel := 0;
   PRODUCT_TYPE[7].Motion.Gluing_Rotary_Jig_Axis.Position[20].Pos := 0;
   PRODUCT_TYPE[7].Motion.Gluing_Rotary_Jig_Axis.Position[20].Vel := 0;
   PRODUCT_TYPE[8].Motion.Gluing_Rotary_Jig_Axis.Position[20].Pos := 0;
   PRODUCT_TYPE[8].Motion.Gluing_Rotary_Jig_Axis.Position[20].Vel := 0;
   PRODUCT_TYPE[9].Motion.Gluing_Rotary_Jig_Axis.Position[20].Pos := 0;
   PRODUCT_TYPE[9].Motion.Gluing_Rotary_Jig_Axis.Position[20].Vel := 0;
   PRODUCT_TYPE[10].Motion.Gluing_Rotary_Jig_Axis.Position[20].Pos := 0;
   PRODUCT_TYPE[10].Motion.Gluing_Rotary_Jig_Axis.Position[20].Vel := 0;
   PRODUCT_TYPE[1].Motion.Ring_Turntable_Axis_2.Position[1].Pos := 3585;
   PRODUCT_TYPE[1].Motion.Ring_Turntable_Axis_2.Position[1].Vel := 10000;
   PRODUCT_TYPE[2].Motion.Ring_Turntable_Axis_2.Position[1].Pos := 3585;
   PRODUCT_TYPE[2].Motion.Ring_Turntable_Axis_2.Position[1].Vel := 10000;
   PRODUCT_TYPE[3].Motion.Ring_Turntable_Axis_2.Position[1].Pos := 3585;
   PRODUCT_TYPE[3].Motion.Ring_Turntable_Axis_2.Position[1].Vel := 10000;
   PRODUCT_TYPE[4].Motion.Ring_Turntable_Axis_2.Position[1].Pos := 3585;
   PRODUCT_TYPE[4].Motion.Ring_Turntable_Axis_2.Position[1].Vel := 10000;
   PRODUCT_TYPE[5].Motion.Ring_Turntable_Axis_2.Position[1].Pos := 3585;
   PRODUCT_TYPE[5].Motion.Ring_Turntable_Axis_2.Position[1].Vel := 10000;
   PRODUCT_TYPE[6].Motion.Ring_Turntable_Axis_2.Position[1].Pos := 3585;
   PRODUCT_TYPE[6].Motion.Ring_Turntable_Axis_2.Position[1].Vel := 10000;
   PRODUCT_TYPE[7].Motion.Ring_Turntable_Axis_2.Position[1].Pos := 3585;
   PRODUCT_TYPE[7].Motion.Ring_Turntable_Axis_2.Position[1].Vel := 10000;
   PRODUCT_TYPE[8].Motion.Ring_Turntable_Axis_2.Position[1].Pos := 3585;
   PRODUCT_TYPE[8].Motion.Ring_Turntable_Axis_2.Position[1].Vel := 10000;
   PRODUCT_TYPE[9].Motion.Ring_Turntable_Axis_2.Position[1].Pos := 3585;
   PRODUCT_TYPE[9].Motion.Ring_Turntable_Axis_2.Position[1].Vel := 10000;
   PRODUCT_TYPE[10].Motion.Ring_Turntable_Axis_2.Position[1].Pos := 3585;
   PRODUCT_TYPE[10].Motion.Ring_Turntable_Axis_2.Position[1].Vel := 10000;
   PRODUCT_TYPE[1].Motion.Ring_Turntable_Axis_2.Position[2].Pos := 48610;
   PRODUCT_TYPE[1].Motion.Ring_Turntable_Axis_2.Position[2].Vel := 10000;
   PRODUCT_TYPE[2].Motion.Ring_Turntable_Axis_2.Position[2].Pos := 48610;
   PRODUCT_TYPE[2].Motion.Ring_Turntable_Axis_2.Position[2].Vel := 10000;
   PRODUCT_TYPE[3].Motion.Ring_Turntable_Axis_2.Position[2].Pos := 48610;
   PRODUCT_TYPE[3].Motion.Ring_Turntable_Axis_2.Position[2].Vel := 10000;
   PRODUCT_TYPE[4].Motion.Ring_Turntable_Axis_2.Position[2].Pos := 48610;
   PRODUCT_TYPE[4].Motion.Ring_Turntable_Axis_2.Position[2].Vel := 10000;
   PRODUCT_TYPE[5].Motion.Ring_Turntable_Axis_2.Position[2].Pos := 48610;
   PRODUCT_TYPE[5].Motion.Ring_Turntable_Axis_2.Position[2].Vel := 10000;
   PRODUCT_TYPE[6].Motion.Ring_Turntable_Axis_2.Position[2].Pos := 48610;
   PRODUCT_TYPE[6].Motion.Ring_Turntable_Axis_2.Position[2].Vel := 10000;
   PRODUCT_TYPE[7].Motion.Ring_Turntable_Axis_2.Position[2].Pos := 48610;
   PRODUCT_TYPE[7].Motion.Ring_Turntable_Axis_2.Position[2].Vel := 10000;
   PRODUCT_TYPE[8].Motion.Ring_Turntable_Axis_2.Position[2].Pos := 48610;
   PRODUCT_TYPE[8].Motion.Ring_Turntable_Axis_2.Position[2].Vel := 10000;
   PRODUCT_TYPE[9].Motion.Ring_Turntable_Axis_2.Position[2].Pos := 48610;
   PRODUCT_TYPE[9].Motion.Ring_Turntable_Axis_2.Position[2].Vel := 10000;
   PRODUCT_TYPE[10].Motion.Ring_Turntable_Axis_2.Position[2].Pos := 48610;
   PRODUCT_TYPE[10].Motion.Ring_Turntable_Axis_2.Position[2].Vel := 10000;
   PRODUCT_TYPE[1].Motion.Ring_Turntable_Axis_2.Position[3].Pos := 93637;
   PRODUCT_TYPE[1].Motion.Ring_Turntable_Axis_2.Position[3].Vel := 10000;
   PRODUCT_TYPE[2].Motion.Ring_Turntable_Axis_2.Position[3].Pos := 93637;
   PRODUCT_TYPE[2].Motion.Ring_Turntable_Axis_2.Position[3].Vel := 10000;
   PRODUCT_TYPE[3].Motion.Ring_Turntable_Axis_2.Position[3].Pos := 93637;
   PRODUCT_TYPE[3].Motion.Ring_Turntable_Axis_2.Position[3].Vel := 10000;
   PRODUCT_TYPE[4].Motion.Ring_Turntable_Axis_2.Position[3].Pos := 93637;
   PRODUCT_TYPE[4].Motion.Ring_Turntable_Axis_2.Position[3].Vel := 10000;
   PRODUCT_TYPE[5].Motion.Ring_Turntable_Axis_2.Position[3].Pos := 93637;
   PRODUCT_TYPE[5].Motion.Ring_Turntable_Axis_2.Position[3].Vel := 10000;
   PRODUCT_TYPE[6].Motion.Ring_Turntable_Axis_2.Position[3].Pos := 93637;
   PRODUCT_TYPE[6].Motion.Ring_Turntable_Axis_2.Position[3].Vel := 10000;
   PRODUCT_TYPE[7].Motion.Ring_Turntable_Axis_2.Position[3].Pos := 93637;
   PRODUCT_TYPE[7].Motion.Ring_Turntable_Axis_2.Position[3].Vel := 10000;
   PRODUCT_TYPE[8].Motion.Ring_Turntable_Axis_2.Position[3].Pos := 93637;
   PRODUCT_TYPE[8].Motion.Ring_Turntable_Axis_2.Position[3].Vel := 10000;
   PRODUCT_TYPE[9].Motion.Ring_Turntable_Axis_2.Position[3].Pos := 93637;
   PRODUCT_TYPE[9].Motion.Ring_Turntable_Axis_2.Position[3].Vel := 10000;
   PRODUCT_TYPE[10].Motion.Ring_Turntable_Axis_2.Position[3].Pos := 93637;
   PRODUCT_TYPE[10].Motion.Ring_Turntable_Axis_2.Position[3].Vel := 10000;
   PRODUCT_TYPE[1].Motion.Ring_Turntable_Axis_2.Position[4].Pos := 138606;
   PRODUCT_TYPE[1].Motion.Ring_Turntable_Axis_2.Position[4].Vel := 10000;
   PRODUCT_TYPE[2].Motion.Ring_Turntable_Axis_2.Position[4].Pos := 138606;
   PRODUCT_TYPE[2].Motion.Ring_Turntable_Axis_2.Position[4].Vel := 10000;
   PRODUCT_TYPE[3].Motion.Ring_Turntable_Axis_2.Position[4].Pos := 138606;
   PRODUCT_TYPE[3].Motion.Ring_Turntable_Axis_2.Position[4].Vel := 10000;
   PRODUCT_TYPE[4].Motion.Ring_Turntable_Axis_2.Position[4].Pos := 138606;
   PRODUCT_TYPE[4].Motion.Ring_Turntable_Axis_2.Position[4].Vel := 10000;
   PRODUCT_TYPE[5].Motion.Ring_Turntable_Axis_2.Position[4].Pos := 138606;
   PRODUCT_TYPE[5].Motion.Ring_Turntable_Axis_2.Position[4].Vel := 10000;
   PRODUCT_TYPE[6].Motion.Ring_Turntable_Axis_2.Position[4].Pos := 138606;
   PRODUCT_TYPE[6].Motion.Ring_Turntable_Axis_2.Position[4].Vel := 10000;
   PRODUCT_TYPE[7].Motion.Ring_Turntable_Axis_2.Position[4].Pos := 138606;
   PRODUCT_TYPE[7].Motion.Ring_Turntable_Axis_2.Position[4].Vel := 10000;
   PRODUCT_TYPE[8].Motion.Ring_Turntable_Axis_2.Position[4].Pos := 138606;
   PRODUCT_TYPE[8].Motion.Ring_Turntable_Axis_2.Position[4].Vel := 10000;
   PRODUCT_TYPE[9].Motion.Ring_Turntable_Axis_2.Position[4].Pos := 138606;
   PRODUCT_TYPE[9].Motion.Ring_Turntable_Axis_2.Position[4].Vel := 10000;
   PRODUCT_TYPE[10].Motion.Ring_Turntable_Axis_2.Position[4].Pos := 138606;
   PRODUCT_TYPE[10].Motion.Ring_Turntable_Axis_2.Position[4].Vel := 10000;
   PRODUCT_TYPE[1].Motion.Ring_Turntable_Axis_2.Position[5].Pos := 183388;
   PRODUCT_TYPE[1].Motion.Ring_Turntable_Axis_2.Position[5].Vel := 10000;
   PRODUCT_TYPE[2].Motion.Ring_Turntable_Axis_2.Position[5].Pos := 183388;
   PRODUCT_TYPE[2].Motion.Ring_Turntable_Axis_2.Position[5].Vel := 10000;
   PRODUCT_TYPE[3].Motion.Ring_Turntable_Axis_2.Position[5].Pos := 183388;
   PRODUCT_TYPE[3].Motion.Ring_Turntable_Axis_2.Position[5].Vel := 10000;
   PRODUCT_TYPE[4].Motion.Ring_Turntable_Axis_2.Position[5].Pos := 183388;
   PRODUCT_TYPE[4].Motion.Ring_Turntable_Axis_2.Position[5].Vel := 10000;
   PRODUCT_TYPE[5].Motion.Ring_Turntable_Axis_2.Position[5].Pos := 183388;
   PRODUCT_TYPE[5].Motion.Ring_Turntable_Axis_2.Position[5].Vel := 10000;
   PRODUCT_TYPE[6].Motion.Ring_Turntable_Axis_2.Position[5].Pos := 183388;
   PRODUCT_TYPE[6].Motion.Ring_Turntable_Axis_2.Position[5].Vel := 10000;
   PRODUCT_TYPE[7].Motion.Ring_Turntable_Axis_2.Position[5].Pos := 183388;
   PRODUCT_TYPE[7].Motion.Ring_Turntable_Axis_2.Position[5].Vel := 10000;
   PRODUCT_TYPE[8].Motion.Ring_Turntable_Axis_2.Position[5].Pos := 183388;
   PRODUCT_TYPE[8].Motion.Ring_Turntable_Axis_2.Position[5].Vel := 10000;
   PRODUCT_TYPE[9].Motion.Ring_Turntable_Axis_2.Position[5].Pos := 183388;
   PRODUCT_TYPE[9].Motion.Ring_Turntable_Axis_2.Position[5].Vel := 10000;
   PRODUCT_TYPE[10].Motion.Ring_Turntable_Axis_2.Position[5].Pos := 183388;
   PRODUCT_TYPE[10].Motion.Ring_Turntable_Axis_2.Position[5].Vel := 10000;
   PRODUCT_TYPE[1].Motion.Ring_Turntable_Axis_2.Position[6].Pos := 228458;
   PRODUCT_TYPE[1].Motion.Ring_Turntable_Axis_2.Position[6].Vel := 10000;
   PRODUCT_TYPE[2].Motion.Ring_Turntable_Axis_2.Position[6].Pos := 228458;
   PRODUCT_TYPE[2].Motion.Ring_Turntable_Axis_2.Position[6].Vel := 10000;
   PRODUCT_TYPE[3].Motion.Ring_Turntable_Axis_2.Position[6].Pos := 228458;
   PRODUCT_TYPE[3].Motion.Ring_Turntable_Axis_2.Position[6].Vel := 10000;
   PRODUCT_TYPE[4].Motion.Ring_Turntable_Axis_2.Position[6].Pos := 228458;
   PRODUCT_TYPE[4].Motion.Ring_Turntable_Axis_2.Position[6].Vel := 10000;
   PRODUCT_TYPE[5].Motion.Ring_Turntable_Axis_2.Position[6].Pos := 228458;
   PRODUCT_TYPE[5].Motion.Ring_Turntable_Axis_2.Position[6].Vel := 10000;
   PRODUCT_TYPE[6].Motion.Ring_Turntable_Axis_2.Position[6].Pos := 228458;
   PRODUCT_TYPE[6].Motion.Ring_Turntable_Axis_2.Position[6].Vel := 10000;
   PRODUCT_TYPE[7].Motion.Ring_Turntable_Axis_2.Position[6].Pos := 228458;
   PRODUCT_TYPE[7].Motion.Ring_Turntable_Axis_2.Position[6].Vel := 10000;
   PRODUCT_TYPE[8].Motion.Ring_Turntable_Axis_2.Position[6].Pos := 228458;
   PRODUCT_TYPE[8].Motion.Ring_Turntable_Axis_2.Position[6].Vel := 10000;
   PRODUCT_TYPE[9].Motion.Ring_Turntable_Axis_2.Position[6].Pos := 228458;
   PRODUCT_TYPE[9].Motion.Ring_Turntable_Axis_2.Position[6].Vel := 10000;
   PRODUCT_TYPE[10].Motion.Ring_Turntable_Axis_2.Position[6].Pos := 228458;
   PRODUCT_TYPE[10].Motion.Ring_Turntable_Axis_2.Position[6].Vel := 10000;
   PRODUCT_TYPE[1].Motion.Ring_Turntable_Axis_2.Position[7].Pos := 273513;
   PRODUCT_TYPE[1].Motion.Ring_Turntable_Axis_2.Position[7].Vel := 10000;
   PRODUCT_TYPE[2].Motion.Ring_Turntable_Axis_2.Position[7].Pos := 273513;
   PRODUCT_TYPE[2].Motion.Ring_Turntable_Axis_2.Position[7].Vel := 10000;
   PRODUCT_TYPE[3].Motion.Ring_Turntable_Axis_2.Position[7].Pos := 273513;
   PRODUCT_TYPE[3].Motion.Ring_Turntable_Axis_2.Position[7].Vel := 10000;
   PRODUCT_TYPE[4].Motion.Ring_Turntable_Axis_2.Position[7].Pos := 273513;
   PRODUCT_TYPE[4].Motion.Ring_Turntable_Axis_2.Position[7].Vel := 10000;
   PRODUCT_TYPE[5].Motion.Ring_Turntable_Axis_2.Position[7].Pos := 273513;
   PRODUCT_TYPE[5].Motion.Ring_Turntable_Axis_2.Position[7].Vel := 10000;
   PRODUCT_TYPE[6].Motion.Ring_Turntable_Axis_2.Position[7].Pos := 273513;
   PRODUCT_TYPE[6].Motion.Ring_Turntable_Axis_2.Position[7].Vel := 10000;
   PRODUCT_TYPE[7].Motion.Ring_Turntable_Axis_2.Position[7].Pos := 273513;
   PRODUCT_TYPE[7].Motion.Ring_Turntable_Axis_2.Position[7].Vel := 10000;
   PRODUCT_TYPE[8].Motion.Ring_Turntable_Axis_2.Position[7].Pos := 273513;
   PRODUCT_TYPE[8].Motion.Ring_Turntable_Axis_2.Position[7].Vel := 10000;
   PRODUCT_TYPE[9].Motion.Ring_Turntable_Axis_2.Position[7].Pos := 273513;
   PRODUCT_TYPE[9].Motion.Ring_Turntable_Axis_2.Position[7].Vel := 10000;
   PRODUCT_TYPE[10].Motion.Ring_Turntable_Axis_2.Position[7].Pos := 273513;
   PRODUCT_TYPE[10].Motion.Ring_Turntable_Axis_2.Position[7].Vel := 10000;
